LIN {X 0,Y 410.552,Z 311.53,A -85,B 0,C 180,E1 -10538.615,E2 -10538.615} C_VEL
LIN {X 0,Y 410.987,Z 304.76,A -85,B 0,C 180,E1 -10540.095,E2 -10540.095} C_VEL
LIN {X 0,Y 411.569,Z 296.376,A -85,B 0,C 180,E1 -10541.575,E2 -10541.575} C_VEL
LIN {X 0,Y 412.223,Z 287.792,A -85,B 0,C 180,E1 -10542.805,E2 -10542.805} C_VEL
LIN {X 0,Y 412.957,Z 277.054,A -85,B 0,C 180,E1 -10544.052,E2 -10544.052} C_VEL
LIN {X 0,Y 413.773,Z 265.358,A -85,B 0,C 180,E1 -10545.138,E2 -10545.138} C_VEL
LIN {X 0,Y 414.618,Z 253.491,A -85,B 0,C 180,E1 -10545.988,E2 -10545.988} C_VEL
LIN {X 0,Y 414.756,Z 247.262,A -85,B 0,C 180,E1 -10546.361,E2 -10546.361} C_VEL
LIN {X 0,Y 412.907,Z 233.741,A -85,B 0,C 180,E1 -10547.084,E2 -10547.084} C_VEL
LIN {X 0,Y 410.788,Z 220.639,A -85,B 0,C 180,E1 -10547.587,E2 -10547.587} C_VEL
LIN {X 0,Y 410.692,Z 219.451,A -85,B 0,C 180,E1 -10547.631,E2 -10547.631} C_VEL
LIN {X 0,Y 411.028,Z 212.027,A -85,B 0,C 180,E1 -10550.519,E2 -10550.519} C_VEL
LIN {X 0,Y 411.452,Z 202.789,A -85,B 0,C 180,E1 -10554.202,E2 -10554.202} C_VEL
LIN {X 0,Y 411.95,Z 194.811,A -85,B 0,C 180,E1 -10557.484,E2 -10557.484} C_VEL
LIN {X 0,Y 412.504,Z 187.23,A -85,B 0,C 180,E1 -10560.739,E2 -10560.739} C_VEL
LIN {X 0,Y 413.051,Z 181.102,A -85,B 0,C 180,E1 -10563.516,E2 -10563.516} C_VEL
LIN {X 0,Y 413.532,Z 176.073,A -85,B 0,C 180,E1 -10565.897,E2 -10565.897} C_VEL
LIN {X 0,Y 413.222,Z 172.446,A -85,B 0,C 180,E1 -10567.755,E2 -10567.755} C_VEL
LIN {X 0,Y 412.08,Z 166.019,A -85,B 0,C 180,E1 -10571.373,E2 -10571.373} C_VEL
LIN {X 0,Y 411.188,Z 161.268,A -85,B 0,C 180,E1 -10574.489,E2 -10574.489} C_VEL
LIN {X 0,Y 411.182,Z 161.271,A -85,B 0,C 180,E1 -10578.195,E2 -10578.195} C_VEL
LIN {X 0,Y 411.226,Z 161.264,A -85,B 0,C 180,E1 -10580.776,E2 -10580.776} C_VEL
LIN {X 0,Y 411.202,Z 161.267,A -85,B 0,C 180,E1 -10584.471,E2 -10584.471} C_VEL
LIN {X 0,Y 411.211,Z 161.265,A -85,B 0,C 180,E1 -10586.873,E2 -10586.873} C_VEL
LIN {X 0,Y 411.237,Z 161.261,A -85,B 0,C 180,E1 -10590.644,E2 -10590.644} C_VEL
LIN {X 0,Y 411.243,Z 161.26,A -85,B 0,C 180,E1 -10593.619,E2 -10593.619} C_VEL
LIN {X 0,Y 411.208,Z 161.264,A -85,B 0,C 180,E1 -10596.852,E2 -10596.852} C_VEL
LIN {X 0,Y 411.219,Z 161.262,A -85,B 0,C 180,E1 -10600.05,E2 -10600.05} C_VEL
LIN {X 0,Y 411.267,Z 161.257,A -85,B 0,C 180,E1 -10603.131,E2 -10603.131} C_VEL
LIN {X 0,Y 411.31,Z 161.252,A -85,B 0,C 180,E1 -10606.895,E2 -10606.895} C_VEL
LIN {X 0,Y 411.298,Z 161.254,A -85,B 0,C 180,E1 -10610.161,E2 -10610.161} C_VEL
LIN {X 0,Y 411.465,Z 161.233,A -85,B 0,C 180,E1 -10613.133,E2 -10613.133} C_VEL
LIN {X 0,Y 411.315,Z 161.251,A -85,B 0,C 180,E1 -10615.099,E2 -10615.099} C_VEL
LIN {X 0,Y 411.519,Z 161.226,A -85,B 0,C 180,E1 -10618.042,E2 -10618.042} C_VEL
LIN {X 0,Y 411.647,Z 161.211,A -85,B 0,C 180,E1 -10619.999,E2 -10619.999} C_VEL
LIN {X 0,Y 411.469,Z 161.234,A -85,B 0,C 180,E1 -10622.937,E2 -10622.937} C_VEL
LIN {X 0,Y 411.45,Z 161.237,A -85,B 0,C 180,E1 -10626.62,E2 -10626.62} C_VEL
LIN {X 0,Y 411.299,Z 161.255,A -85,B 0,C 180,E1 -10628.846,E2 -10628.846} C_VEL
LIN {X 0,Y 411.065,Z 161.351,A -85,B 0,C 180,E1 -10630.84,E2 -10630.84} C_VEL
LIN {X 0,Y 411.063,Z 163.277,A -85,B 0,C 180,E1 -10632.956,E2 -10632.956} C_VEL
LIN {X 0,Y 410.89,Z 166.763,A -85,B 0,C 180,E1 -10636.695,E2 -10636.695} C_VEL
LIN {X 0,Y 410.695,Z 169.909,A -85,B 0,C 180,E1 -10640.013,E2 -10640.013} C_VEL
LIN {X 0,Y 410.604,Z 172.966,A -85,B 0,C 180,E1 -10643.183,E2 -10643.183} C_VEL
LIN {X 0,Y 410.501,Z 176.153,A -85,B 0,C 180,E1 -10646.431,E2 -10646.431} C_VEL
LIN {X 0,Y 410.553,Z 177.376,A -85,B 0,C 180,E1 -10647.491,E2 -10647.491} C_VEL
LIN {X 0,Y 414.209,Z 190.782,A -85,B 0,C 180,E1 -10648.157,E2 -10648.157} C_VEL
LIN {X 0,Y 415.754,Z 198.207,A -85,B 0,C 180,E1 -10648.593,E2 -10648.593} C_VEL
LIN {X 0,Y 415.142,Z 210.294,A -85,B 0,C 180,E1 -10649.333,E2 -10649.333} C_VEL
LIN {X 0,Y 414.416,Z 221.682,A -85,B 0,C 180,E1 -10650.233,E2 -10650.233} C_VEL
LIN {X 0,Y 413.716,Z 232.745,A -85,B 0,C 180,E1 -10651.345,E2 -10651.345} C_VEL
LIN {X 0,Y 412.965,Z 242.44,A -85,B 0,C 180,E1 -10652.561,E2 -10652.561} C_VEL
LIN {X 0,Y 412.328,Z 250.391,A -85,B 0,C 180,E1 -10653.778,E2 -10653.778} C_VEL
LIN {X 0,Y 411.629,Z 257.985,A -85,B 0,C 180,E1 -10655.195,E2 -10655.195} C_VEL
LIN {X 0,Y 411.155,Z 264.595,A -85,B 0,C 180,E1 -10656.745,E2 -10656.745} C_VEL
LIN {X 0,Y 410.782,Z 269.178,A -85,B 0,C 180,E1 -10658.093,E2 -10658.093} C_VEL
LIN {X 0,Y 410.457,Z 273.169,A -85,B 0,C 180,E1 -10659.6,E2 -10659.6} C_VEL
LIN {X 0,Y 410.255,Z 276.038,A -85,B 0,C 180,E1 -10661.083,E2 -10661.083} C_VEL
LIN {X 0,Y 410.05,Z 277.889,A -85,B 0,C 180,E1 -10662.524,E2 -10662.524} C_VEL
LIN {X 0,Y 409.999,Z 278.849,A -85,B 0,C 180,E1 -10663.95,E2 -10663.95} C_VEL
LIN {X 0,Y 409.939,Z 278.987,A -85,B 0,C 180,E1 -10665.339,E2 -10665.339} C_VEL
LIN {X 0,Y 409.979,Z 278.355,A -85,B 0,C 180,E1 -10666.709,E2 -10666.709} C_VEL
LIN {X 0,Y 410.11,Z 276.96,A -85,B 0,C 180,E1 -10668.061,E2 -10668.061} C_VEL
LIN {X 0,Y 410.276,Z 274.799,A -85,B 0,C 180,E1 -10669.387,E2 -10669.387} C_VEL
LIN {X 0,Y 410.447,Z 271.931,A -85,B 0,C 180,E1 -10670.688,E2 -10670.688} C_VEL
LIN {X 0,Y 410.795,Z 267.236,A -85,B 0,C 180,E1 -10672.293,E2 -10672.293} C_VEL
LIN {X 0,Y 411.226,Z 260.795,A -85,B 0,C 180,E1 -10673.981,E2 -10673.981} C_VEL
LIN {X 0,Y 411.688,Z 253.986,A -85,B 0,C 180,E1 -10675.387,E2 -10675.387} C_VEL
LIN {X 0,Y 412.342,Z 246.022,A -85,B 0,C 180,E1 -10676.723,E2 -10676.723} C_VEL
LIN {X 0,Y 413.027,Z 236.553,A -85,B 0,C 180,E1 -10678.02,E2 -10678.02} C_VEL
LIN {X 0,Y 413.582,Z 227.231,A -85,B 0,C 180,E1 -10679.067,E2 -10679.067} C_VEL
LIN {X 0,Y 414.269,Z 215.745,A -85,B 0,C 180,E1 -10680.102,E2 -10680.102} C_VEL
LIN {X 0,Y 414.955,Z 203.945,A -85,B 0,C 180,E1 -10680.93,E2 -10680.93} C_VEL
LIN {X 0,Y 415.343,Z 197.322,A -85,B 0,C 180,E1 -10681.306,E2 -10681.306} C_VEL
LIN {X 0,Y 412.71,Z 185.249,A -85,B 0,C 180,E1 -10681.972,E2 -10681.972} C_VEL
LIN {X 0,Y 410.376,Z 175.545,A -85,B 0,C 180,E1 -10682.389,E2 -10682.389} C_VEL
LIN {X 0,Y 410.392,Z 171.916,A -85,B 0,C 180,E1 -10685.732,E2 -10685.732} C_VEL
LIN {X 0,Y 410.404,Z 168.584,A -85,B 0,C 180,E1 -10688.923,E2 -10688.923} C_VEL
LIN {X 0,Y 410.492,Z 165.336,A -85,B 0,C 180,E1 -10692.05,E2 -10692.05} C_VEL
LIN {X 0,Y 410.643,Z 162.203,A -85,B 0,C 180,E1 -10695.124,E2 -10695.124} C_VEL
LIN {X 0,Y 410.668,Z 161.335,A -85,B 0,C 180,E1 -10696.137,E2 -10696.137} C_VEL
LIN {X 0,Y 411.106,Z 161.275,A -85,B 0,C 180,E1 -10699.161,E2 -10699.161} C_VEL
LIN {X 0,Y 411.434,Z 161.237,A -85,B 0,C 180,E1 -10702.191,E2 -10702.191} C_VEL
LIN {X 0,Y 411.461,Z 161.234,A -85,B 0,C 180,E1 -10704.118,E2 -10704.118} C_VEL
LIN {X 0,Y 411.511,Z 161.228,A -85,B 0,C 180,E1 -10708.042,E2 -10708.042} C_VEL
LIN {X 0,Y 411.639,Z 161.213,A -85,B 0,C 180,E1 -10710,E2 -10710} C_VEL
LIN {X 0,Y 411.463,Z 161.229,A -85,B 0,C 180,E1 -10712.937,E2 -10712.937} C_VEL
LIN {X 0,Y 411.325,Z 161.247,A -85,B 0,C 180,E1 -10713.48,E2 -10713.48} C_VEL
LIN {X 0,Y 410.551,Z 161.347,A -85,B 0,C 180,E1 -10714.298,E2 -10714.298} C_VEL
LIN {X 0,Y 407.721,Z 161.699,A -85,B 0,C 180,E1 -10715.629,E2 -10715.629} C_VEL
LIN {X 0,Y 405.424,Z 161.983,A -85,B 0,C 180,E1 -10716.704,E2 -10716.704} C_VEL
LIN {X 0,Y 404.482,Z 162.103,A -85,B 0,C 180,E1 -10717.533,E2 -10717.533} C_VEL
LIN {X 0,Y 404.423,Z 162.11,A -85,B 0,C 180,E1 -10717.813,E2 -10717.813} C_VEL
LIN {X 0,Y 404.253,Z 162.131,A -85,B 0,C 180,E1 -10722.041,E2 -10722.041} C_VEL
LIN {X 0,Y 404.203,Z 162.136,A -85,B 0,C 180,E1 -10725.118,E2 -10725.118} C_VEL
LIN {X 0,Y 404.207,Z 162.134,A -85,B 0,C 180,E1 -10728.238,E2 -10728.238} C_VEL
LIN {X 0,Y 404.136,Z 162.146,A -85,B 0,C 180,E1 -10731.419,E2 -10731.419} C_VEL
LIN {X 0,Y 404.174,Z 162.138,A -85,B 0,C 180,E1 -10734.666,E2 -10734.666} C_VEL
LIN {X 0,Y 404.192,Z 162.136,A -85,B 0,C 180,E1 -10738,E2 -10738} C_VEL
LIN {X 0,Y 404.136,Z 162.146,A -85,B 0,C 180,E1 -10741.558,E2 -10741.558} C_VEL
LIN {X 0,Y 404.181,Z 162.14,A -85,B 0,C 180,E1 -10745.016,E2 -10745.016} C_VEL
LIN {X 0,Y 404.153,Z 162.143,A -85,B 0,C 180,E1 -10748.757,E2 -10748.757} C_VEL
LIN {X 0,Y 404.121,Z 162.147,A -85,B 0,C 180,E1 -10751.6,E2 -10751.6} C_VEL
LIN {X 0,Y 404.146,Z 162.142,A -85,B 0,C 180,E1 -10754.523,E2 -10754.523} C_VEL
LIN {X 0,Y 404.134,Z 162.146,A -85,B 0,C 180,E1 -10757.296,E2 -10757.296} C_VEL
LIN {X 0,Y 404.166,Z 162.139,A -85,B 0,C 180,E1 -10759.956,E2 -10759.956} C_VEL
LIN {X 0,Y 404.138,Z 162.145,A -85,B 0,C 180,E1 -10763.125,E2 -10763.125} C_VEL
LIN {X 0,Y 404.143,Z 162.143,A -85,B 0,C 180,E1 -10766.188,E2 -10766.188} C_VEL
LIN {X 0,Y 404.144,Z 162.141,A -85,B 0,C 180,E1 -10769.715,E2 -10769.715} C_VEL
LIN {X 0,Y 404.194,Z 162.137,A -85,B 0,C 180,E1 -10773.123,E2 -10773.123} C_VEL
LIN {X 0,Y 404.176,Z 162.138,A -85,B 0,C 180,E1 -10775.335,E2 -10775.335} C_VEL
LIN {X 0,Y 404.159,Z 162.144,A -85,B 0,C 180,E1 -10778.582,E2 -10778.582} C_VEL
LIN {X 0,Y 404.208,Z 162.135,A -85,B 0,C 180,E1 -10781.762,E2 -10781.762} C_VEL
LIN {X 0,Y 404.206,Z 162.135,A -85,B 0,C 180,E1 -10784.883,E2 -10784.883} C_VEL
LIN {X 0,Y 404.257,Z 162.13,A -85,B 0,C 180,E1 -10787.959,E2 -10787.959} C_VEL
LIN {X 0,Y 404.404,Z 162.114,A -85,B 0,C 180,E1 -10792.131,E2 -10792.131} C_VEL
LIN {X 0,Y 404.419,Z 162.111,A -85,B 0,C 180,E1 -10794.016,E2 -10794.016} C_VEL
LIN {X 0,Y 404.484,Z 162.103,A -85,B 0,C 180,E1 -10798.009,E2 -10798.009} C_VEL
LIN {X 0,Y 404.611,Z 162.087,A -85,B 0,C 180,E1 -10800.001,E2 -10800.001} C_VEL
LIN {X 0,Y 404.417,Z 162.108,A -85,B 0,C 180,E1 -10802.989,E2 -10802.989} C_VEL
LIN {X 0,Y 404.371,Z 162.113,A -85,B 0,C 180,E1 -10806.988,E2 -10806.988} C_VEL
LIN {X 0,Y 404.259,Z 162.131,A -85,B 0,C 180,E1 -10810.012,E2 -10810.012} C_VEL
LIN {X 0,Y 404.268,Z 162.128,A -85,B 0,C 180,E1 -10813.212,E2 -10813.212} C_VEL
LIN {X 0,Y 404.218,Z 162.133,A -85,B 0,C 180,E1 -10817.007,E2 -10817.007} C_VEL
LIN {X 0,Y 404.166,Z 162.139,A -85,B 0,C 180,E1 -10820.352,E2 -10820.352} C_VEL
LIN {X 0,Y 404.172,Z 162.142,A -85,B 0,C 180,E1 -10823.575,E2 -10823.575} C_VEL
LIN {X 0,Y 404.186,Z 162.139,A -85,B 0,C 180,E1 -10825.767,E2 -10825.767} C_VEL
LIN {X 0,Y 404.197,Z 162.137,A -85,B 0,C 180,E1 -10828,E2 -10828} C_VEL
LIN {X 0,Y 404.141,Z 162.146,A -85,B 0,C 180,E1 -10831.558,E2 -10831.558} C_VEL
LIN {X 0,Y 404.186,Z 162.14,A -85,B 0,C 180,E1 -10835.017,E2 -10835.017} C_VEL
LIN {X 0,Y 404.155,Z 162.142,A -85,B 0,C 180,E1 -10838.757,E2 -10838.757} C_VEL
LIN {X 0,Y 404.125,Z 162.146,A -85,B 0,C 180,E1 -10841.6,E2 -10841.6} C_VEL
LIN {X 0,Y 404.148,Z 162.138,A -85,B 0,C 180,E1 -10844.522,E2 -10844.522} C_VEL
LIN {X 0,Y 404.174,Z 162.299,A -85,B 0,C 180,E1 -10846.103,E2 -10846.103} C_VEL
LIN {X 0,Y 405.082,Z 167.107,A -85,B 0,C 180,E1 -10848.755,E2 -10848.755} C_VEL
LIN {X 0,Y 406.218,Z 173.548,A -85,B 0,C 180,E1 -10852.108,E2 -10852.108} C_VEL
LIN {X 0,Y 406.527,Z 177.404,A -85,B 0,C 180,E1 -10854,E2 -10854} C_VEL
LIN {X 0,Y 406.009,Z 183.846,A -85,B 0,C 180,E1 -10856.957,E2 -10856.957} C_VEL
LIN {X 0,Y 405.458,Z 190.289,A -85,B 0,C 180,E1 -10859.823,E2 -10859.823} C_VEL
LIN {X 0,Y 404.993,Z 196.978,A -85,B 0,C 180,E1 -10862.704,E2 -10862.704} C_VEL
LIN {X 0,Y 404.383,Z 205.889,A -85,B 0,C 180,E1 -10866.439,E2 -10866.439} C_VEL
LIN {X 0,Y 403.91,Z 214.589,A -85,B 0,C 180,E1 -10869.985,E2 -10869.985} C_VEL
LIN {X 0,Y 403.652,Z 219.873,A -85,B 0,C 180,E1 -10872.097,E2 -10872.097} C_VEL
LIN {X 0,Y 405.923,Z 233.642,A -85,B 0,C 180,E1 -10872.623,E2 -10872.623} C_VEL
LIN {X 0,Y 407.729,Z 246.619,A -85,B 0,C 180,E1 -10873.319,E2 -10873.319} C_VEL
LIN {X 0,Y 407.879,Z 251.732,A -85,B 0,C 180,E1 -10873.631,E2 -10873.631} C_VEL
LIN {X 0,Y 407.03,Z 263.745,A -85,B 0,C 180,E1 -10874.477,E2 -10874.477} C_VEL
LIN {X 0,Y 406.19,Z 275.278,A -85,B 0,C 180,E1 -10875.522,E2 -10875.522} C_VEL
LIN {X 0,Y 405.413,Z 285.747,A -85,B 0,C 180,E1 -10876.721,E2 -10876.721} C_VEL
LIN {X 0,Y 404.71,Z 294.651,A -85,B 0,C 180,E1 -10877.972,E2 -10877.972} C_VEL
LIN {X 0,Y 404.038,Z 303.354,A -85,B 0,C 180,E1 -10879.476,E2 -10879.476} C_VEL
LIN {X 0,Y 403.575,Z 310.309,A -85,B 0,C 180,E1 -10880.983,E2 -10880.983} C_VEL
LIN {X 0,Y 403.204,Z 315.883,A -85,B 0,C 180,E1 -10882.488,E2 -10882.488} C_VEL
LIN {X 0,Y 403.016,Z 320.261,A -85,B 0,C 180,E1 -10883.994,E2 -10883.994} C_VEL
LIN {X 0,Y 403.002,Z 322.579,A -85,B 0,C 180,E1 -10884.998,E2 -10884.998} C_VEL
LIN {X 0,Y 402.876,Z 324.452,A -85,B 0,C 180,E1 -10885.999,E2 -10885.999} C_VEL
LIN {X 0,Y 402.895,Z 325.862,A -85,B 0,C 180,E1 -10887,E2 -10887} C_VEL
LIN {X 0,Y 402.92,Z 326.863,A -85,B 0,C 180,E1 -10888.001,E2 -10888.001} C_VEL
LIN {X 0,Y 402.879,Z 327.673,A -85,B 0,C 180,E1 -10890,E2 -10890} C_VEL
LIN {X 0,Y 402.875,Z 327.442,A -85,B 0,C 180,E1 -10891,E2 -10891} C_VEL
LIN {X 0,Y 402.922,Z 326.814,A -85,B 0,C 180,E1 -10891.999,E2 -10891.999} C_VEL
LIN {X 0,Y 402.909,Z 325.788,A -85,B 0,C 180,E1 -10893,E2 -10893} C_VEL
LIN {X 0,Y 402.878,Z 324.353,A -85,B 0,C 180,E1 -10894.001,E2 -10894.001} C_VEL
LIN {X 0,Y 403.007,Z 321.356,A -85,B 0,C 180,E1 -10895.504,E2 -10895.504} C_VEL
LIN {X 0,Y 403.118,Z 317.303,A -85,B 0,C 180,E1 -10897.01,E2 -10897.01} C_VEL
LIN {X 0,Y 403.518,Z 311.093,A -85,B 0,C 180,E1 -10898.766,E2 -10898.766} C_VEL
LIN {X 0,Y 403.962,Z 304.323,A -85,B 0,C 180,E1 -10900.272,E2 -10900.272} C_VEL
LIN {X 0,Y 404.576,Z 295.944,A -85,B 0,C 180,E1 -10901.778,E2 -10901.778} C_VEL
LIN {X 0,Y 405.244,Z 287.368,A -85,B 0,C 180,E1 -10903.03,E2 -10903.03} C_VEL
LIN {X 0,Y 405.982,Z 277.521,A -85,B 0,C 180,E1 -10904.204,E2 -10904.204} C_VEL
LIN {X 0,Y 406.781,Z 266.392,A -85,B 0,C 180,E1 -10905.277,E2 -10905.277} C_VEL
LIN {X 0,Y 407.649,Z 255.13,A -85,B 0,C 180,E1 -10906.134,E2 -10906.134} C_VEL
LIN {X 0,Y 407.91,Z 248.55,A -85,B 0,C 180,E1 -10906.55,E2 -10906.55} C_VEL
LIN {X 0,Y 406.128,Z 235.006,A -85,B 0,C 180,E1 -10907.314,E2 -10907.314} C_VEL
LIN {X 0,Y 404.092,Z 222.004,A -85,B 0,C 180,E1 -10907.858,E2 -10907.858} C_VEL
LIN {X 0,Y 403.633,Z 218.99,A -85,B 0,C 180,E1 -10907.97,E2 -10907.97} C_VEL
LIN {X 0,Y 403.958,Z 211.643,A -85,B 0,C 180,E1 -10910.895,E2 -10910.895} C_VEL
LIN {X 0,Y 404.447,Z 202.456,A -85,B 0,C 180,E1 -10914.648,E2 -10914.648} C_VEL
LIN {X 0,Y 404.985,Z 194.699,A -85,B 0,C 180,E1 -10917.941,E2 -10917.941} C_VEL
LIN {X 0,Y 405.601,Z 187.044,A -85,B 0,C 180,E1 -10921.321,E2 -10921.321} C_VEL
LIN {X 0,Y 406.306,Z 179.599,A -85,B 0,C 180,E1 -10924.807,E2 -10924.807} C_VEL
LIN {X 0,Y 406.507,Z 175.952,A -85,B 0,C 180,E1 -10926.617,E2 -10926.617} C_VEL
LIN {X 0,Y 405.925,Z 171.895,A -85,B 0,C 180,E1 -10928.82,E2 -10928.82} C_VEL
LIN {X 0,Y 405.039,Z 166.908,A -85,B 0,C 180,E1 -10931.745,E2 -10931.745} C_VEL
LIN {X 0,Y 404.129,Z 162.148,A -85,B 0,C 180,E1 -10934.912,E2 -10934.912} C_VEL
LIN {X 0,Y 404.141,Z 162.149,A -85,B 0,C 180,E1 -10937.296,E2 -10937.296} C_VEL
LIN {X 0,Y 404.173,Z 162.145,A -85,B 0,C 180,E1 -10939.955,E2 -10939.955} C_VEL
LIN {X 0,Y 404.141,Z 162.147,A -85,B 0,C 180,E1 -10943.125,E2 -10943.125} C_VEL
LIN {X 0,Y 404.149,Z 162.144,A -85,B 0,C 180,E1 -10946.188,E2 -10946.188} C_VEL
LIN {X 0,Y 404.15,Z 162.144,A -85,B 0,C 180,E1 -10949.715,E2 -10949.715} C_VEL
LIN {X 0,Y 404.2,Z 162.136,A -85,B 0,C 180,E1 -10953.123,E2 -10953.123} C_VEL
LIN {X 0,Y 404.182,Z 162.138,A -85,B 0,C 180,E1 -10955.334,E2 -10955.334} C_VEL
LIN {X 0,Y 404.143,Z 162.146,A -85,B 0,C 180,E1 -10958.58,E2 -10958.58} C_VEL
LIN {X 0,Y 404.209,Z 162.133,A -85,B 0,C 180,E1 -10961.761,E2 -10961.761} C_VEL
LIN {X 0,Y 404.211,Z 162.136,A -85,B 0,C 180,E1 -10964.882,E2 -10964.882} C_VEL
LIN {X 0,Y 404.261,Z 162.13,A -85,B 0,C 180,E1 -10967.958,E2 -10967.958} C_VEL
LIN {X 0,Y 404.438,Z 162.108,A -85,B 0,C 180,E1 -10972.099,E2 -10972.099} C_VEL
LIN {X 0,Y 404.428,Z 162.109,A -85,B 0,C 180,E1 -10974.015,E2 -10974.015} C_VEL
LIN {X 0,Y 404.487,Z 162.102,A -85,B 0,C 180,E1 -10978.008,E2 -10978.008} C_VEL
LIN {X 0,Y 404.616,Z 162.087,A -85,B 0,C 180,E1 -10979.999,E2 -10979.999} C_VEL
LIN {X 0,Y 404.426,Z 162.111,A -85,B 0,C 180,E1 -10982.988,E2 -10982.988} C_VEL
LIN {X 0,Y 404.395,Z 162.115,A -85,B 0,C 180,E1 -10986.619,E2 -10986.619} C_VEL
LIN {X 0,Y 404.239,Z 162.134,A -85,B 0,C 180,E1 -10989.002,E2 -10989.002} C_VEL
LIN {X 0,Y 404.05,Z 162.548,A -85,B 0,C 180,E1 -10991.03,E2 -10991.03} C_VEL
LIN {X 0,Y 403.942,Z 165.314,A -85,B 0,C 180,E1 -10994.097,E2 -10994.097} C_VEL
LIN {X 0,Y 403.8,Z 168.179,A -85,B 0,C 180,E1 -10997.21,E2 -10997.21} C_VEL
LIN {X 0,Y 403.637,Z 171.148,A -85,B 0,C 180,E1 -11000.379,E2 -11000.379} C_VEL
LIN {X 0,Y 403.533,Z 174.235,A -85,B 0,C 180,E1 -11003.613,E2 -11003.613} C_VEL
LIN {X 0,Y 403.457,Z 177.672,A -85,B 0,C 180,E1 -11007.138,E2 -11007.138} C_VEL
LIN {X 0,Y 407.287,Z 191.331,A -85,B 0,C 180,E1 -11007.845,E2 -11007.845} C_VEL
LIN {X 0,Y 408.819,Z 198.299,A -85,B 0,C 180,E1 -11008.268,E2 -11008.268} C_VEL
LIN {X 0,Y 408.404,Z 210.267,A -85,B 0,C 180,E1 -11009.016,E2 -11009.016} C_VEL
LIN {X 0,Y 407.575,Z 222.551,A -85,B 0,C 180,E1 -11010.003,E2 -11010.003} C_VEL
LIN {X 0,Y 406.873,Z 233.199,A -85,B 0,C 180,E1 -11011.097,E2 -11011.097} C_VEL
LIN {X 0,Y 406.159,Z 241.938,A -85,B 0,C 180,E1 -11012.197,E2 -11012.197} C_VEL
LIN {X 0,Y 405.346,Z 251.431,A -85,B 0,C 180,E1 -11013.67,E2 -11013.67} C_VEL
LIN {X 0,Y 404.561,Z 259.614,A -85,B 0,C 180,E1 -11015.265,E2 -11015.265} C_VEL
LIN {X 0,Y 404.076,Z 266.026,A -85,B 0,C 180,E1 -11016.863,E2 -11016.863} C_VEL
LIN {X 0,Y 403.659,Z 270.92,A -85,B 0,C 180,E1 -11018.419,E2 -11018.419} C_VEL
LIN {X 0,Y 403.308,Z 274.978,A -85,B 0,C 180,E1 -11020.147,E2 -11020.147} C_VEL
LIN {X 0,Y 403.125,Z 277.173,A -85,B 0,C 180,E1 -11021.489,E2 -11021.489} C_VEL
LIN {X 0,Y 402.937,Z 278.69,A -85,B 0,C 180,E1 -11022.898,E2 -11022.898} C_VEL
LIN {X 0,Y 402.879,Z 279.416,A -85,B 0,C 180,E1 -11024.338,E2 -11024.338} C_VEL
LIN {X 0,Y 402.864,Z 279.33,A -85,B 0,C 180,E1 -11025.749,E2 -11025.749} C_VEL
LIN {X 0,Y 402.937,Z 278.433,A -85,B 0,C 180,E1 -11027.138,E2 -11027.138} C_VEL
LIN {X 0,Y 403.094,Z 276.709,A -85,B 0,C 180,E1 -11028.564,E2 -11028.564} C_VEL
LIN {X 0,Y 403.296,Z 273.981,A -85,B 0,C 180,E1 -11030.063,E2 -11030.063} C_VEL
LIN {X 0,Y 403.55,Z 270.13,A -85,B 0,C 180,E1 -11031.599,E2 -11031.599} C_VEL
LIN {X 0,Y 403.924,Z 264.993,A -85,B 0,C 180,E1 -11033.164,E2 -11033.164} C_VEL
LIN {X 0,Y 404.415,Z 258.326,A -85,B 0,C 180,E1 -11034.762,E2 -11034.762} C_VEL
LIN {X 0,Y 405.074,Z 249.676,A -85,B 0,C 180,E1 -11036.386,E2 -11036.386} C_VEL
LIN {X 0,Y 405.865,Z 240.146,A -85,B 0,C 180,E1 -11037.816,E2 -11037.816} C_VEL
LIN {X 0,Y 406.542,Z 230.234,A -85,B 0,C 180,E1 -11039.011,E2 -11039.011} C_VEL
LIN {X 0,Y 407.239,Z 218.894,A -85,B 0,C 180,E1 -11040.111,E2 -11040.111} C_VEL
LIN {X 0,Y 408,Z 206.876,A -85,B 0,C 180,E1 -11041.022,E2 -11041.022} C_VEL
LIN {X 0,Y 408.289,Z 197.054,A -85,B 0,C 180,E1 -11041.612,E2 -11041.612} C_VEL
LIN {X 0,Y 405.302,Z 183.991,A -85,B 0,C 180,E1 -11042.329,E2 -11042.329} C_VEL
LIN {X 0,Y 403.301,Z 175.836,A -85,B 0,C 180,E1 -11042.713,E2 -11042.713} C_VEL
LIN {X 0,Y 403.374,Z 173.101,A -85,B 0,C 180,E1 -11045.282,E2 -11045.282} C_VEL
LIN {X 0,Y 403.32,Z 169.729,A -85,B 0,C 180,E1 -11048.535,E2 -11048.535} C_VEL
LIN {X 0,Y 403.441,Z 166.434,A -85,B 0,C 180,E1 -11051.726,E2 -11051.726} C_VEL
LIN {X 0,Y 403.567,Z 163.266,A -85,B 0,C 180,E1 -11054.857,E2 -11054.857} C_VEL
LIN {X 0,Y 403.584,Z 162.249,A -85,B 0,C 180,E1 -11055.889,E2 -11055.889} C_VEL
LIN {X 0,Y 404.027,Z 162.157,A -85,B 0,C 180,E1 -11058.969,E2 -11058.969} C_VEL
LIN {X 0,Y 404.374,Z 162.117,A -85,B 0,C 180,E1 -11062.157,E2 -11062.157} C_VEL
LIN {X 0,Y 404.408,Z 162.113,A -85,B 0,C 180,E1 -11064.015,E2 -11064.015} C_VEL
LIN {X 0,Y 404.48,Z 162.104,A -85,B 0,C 180,E1 -11068.008,E2 -11068.008} C_VEL
LIN {X 0,Y 404.608,Z 162.089,A -85,B 0,C 180,E1 -11070,E2 -11070} C_VEL
LIN {X 0,Y 404.42,Z 162.107,A -85,B 0,C 180,E1 -11072.988,E2 -11072.988} C_VEL
LIN {X 0,Y 404.406,Z 162.109,A -85,B 0,C 180,E1 -11076.987,E2 -11076.987} C_VEL
LIN {X 0,Y 404.423,Z 162.11,A -85,B 0,C 180,E1 -11077.813,E2 -11077.813} C_VEL
LIN {X 0,Y 403.774,Z 162.195,A -85,B 0,C 180,E1 -11078.644,E2 -11078.644} C_VEL
LIN {X 0,Y 400.822,Z 162.56,A -85,B 0,C 180,E1 -11079.99,E2 -11079.99} C_VEL
LIN {X 0,Y 398.32,Z 162.868,A -85,B 0,C 180,E1 -11081.078,E2 -11081.078} C_VEL
LIN {X 0,Y 397.278,Z 163.001,A -85,B 0,C 180,E1 -11081.921,E2 -11081.921} C_VEL
LIN {X 0,Y 397.212,Z 163.006,A -85,B 0,C 180,E1 -11082.207,E2 -11082.207} C_VEL
LIN {X 0,Y 397.176,Z 163.012,A -85,B 0,C 180,E1 -11085.392,E2 -11085.392} C_VEL
LIN {X 0,Y 397.159,Z 163.011,A -85,B 0,C 180,E1 -11088.573,E2 -11088.573} C_VEL
LIN {X 0,Y 397.094,Z 163.023,A -85,B 0,C 180,E1 -11091.819,E2 -11091.819} C_VEL
LIN {X 0,Y 397.153,Z 163.015,A -85,B 0,C 180,E1 -11095.132,E2 -11095.132} C_VEL
LIN {X 0,Y 397.158,Z 163.014,A -85,B 0,C 180,E1 -11097.776,E2 -11097.776} C_VEL
LIN {X 0,Y 397.075,Z 163.024,A -85,B 0,C 180,E1 -11100.883,E2 -11100.883} C_VEL
LIN {X 0,Y 397.122,Z 163.016,A -85,B 0,C 180,E1 -11104.494,E2 -11104.494} C_VEL
LIN {X 0,Y 397.1,Z 163.019,A -85,B 0,C 180,E1 -11108.275,E2 -11108.275} C_VEL
LIN {X 0,Y 397.086,Z 163.024,A -85,B 0,C 180,E1 -11110.909,E2 -11110.909} C_VEL
LIN {X 0,Y 397.101,Z 163.02,A -85,B 0,C 180,E1 -11113.648,E2 -11113.648} C_VEL
LIN {X 0,Y 397.1,Z 163.021,A -85,B 0,C 180,E1 -11116.521,E2 -11116.521} C_VEL
LIN {X 0,Y 397.112,Z 163.019,A -85,B 0,C 180,E1 -11120.423,E2 -11120.423} C_VEL
LIN {X 0,Y 397.107,Z 163.019,A -85,B 0,C 180,E1 -11124.266,E2 -11124.266} C_VEL
LIN {X 0,Y 397.113,Z 163.022,A -85,B 0,C 180,E1 -11126.728,E2 -11126.728} C_VEL
LIN {X 0,Y 397.123,Z 163.018,A -85,B 0,C 180,E1 -11130.296,E2 -11130.296} C_VEL
LIN {X 0,Y 397.193,Z 163.012,A -85,B 0,C 180,E1 -11132.61,E2 -11132.61} C_VEL
LIN {X 0,Y 397.132,Z 163.016,A -85,B 0,C 180,E1 -11135.982,E2 -11135.982} C_VEL
LIN {X 0,Y 397.138,Z 163.014,A -85,B 0,C 180,E1 -11139.705,E2 -11139.705} C_VEL
LIN {X 0,Y 397.182,Z 163.011,A -85,B 0,C 180,E1 -11142.845,E2 -11142.845} C_VEL
LIN {X 0,Y 397.229,Z 163.006,A -85,B 0,C 180,E1 -11146.703,E2 -11146.703} C_VEL
LIN {X 0,Y 397.218,Z 163.006,A -85,B 0,C 180,E1 -11149.81,E2 -11149.81} C_VEL
LIN {X 0,Y 397.343,Z 162.99,A -85,B 0,C 180,E1 -11152.888,E2 -11152.888} C_VEL
LIN {X 0,Y 397.255,Z 163,A -85,B 0,C 180,E1 -11154.926,E2 -11154.926} C_VEL
LIN {X 0,Y 397.453,Z 162.979,A -85,B 0,C 180,E1 -11157.974,E2 -11157.974} C_VEL
LIN {X 0,Y 397.58,Z 162.963,A -85,B 0,C 180,E1 -11160.001,E2 -11160.001} C_VEL
LIN {X 0,Y 397.377,Z 162.985,A -85,B 0,C 180,E1 -11163.042,E2 -11163.042} C_VEL
LIN {X 0,Y 397.347,Z 162.992,A -85,B 0,C 180,E1 -11166.092,E2 -11166.092} C_VEL
LIN {X 0,Y 397.237,Z 163.003,A -85,B 0,C 180,E1 -11169.163,E2 -11169.163} C_VEL
LIN {X 0,Y 397.221,Z 163.006,A -85,B 0,C 180,E1 -11172.259,E2 -11172.259} C_VEL
LIN {X 0,Y 397.181,Z 163.012,A -85,B 0,C 180,E1 -11175.392,E2 -11175.392} C_VEL
LIN {X 0,Y 397.164,Z 163.011,A -85,B 0,C 180,E1 -11178.574,E2 -11178.574} C_VEL
LIN {X 0,Y 397.099,Z 163.023,A -85,B 0,C 180,E1 -11181.819,E2 -11181.819} C_VEL
LIN {X 0,Y 397.159,Z 163.015,A -85,B 0,C 180,E1 -11185.132,E2 -11185.132} C_VEL
LIN {X 0,Y 397.164,Z 163.014,A -85,B 0,C 180,E1 -11187.776,E2 -11187.776} C_VEL
LIN {X 0,Y 397.081,Z 163.023,A -85,B 0,C 180,E1 -11190.883,E2 -11190.883} C_VEL
LIN {X 0,Y 397.127,Z 163.016,A -85,B 0,C 180,E1 -11194.494,E2 -11194.494} C_VEL
LIN {X 0,Y 397.103,Z 163.021,A -85,B 0,C 180,E1 -11198.275,E2 -11198.275} C_VEL
LIN {X 0,Y 397.091,Z 163.024,A -85,B 0,C 180,E1 -11200.909,E2 -11200.909} C_VEL
LIN {X 0,Y 397.103,Z 163.017,A -85,B 0,C 180,E1 -11203.649,E2 -11203.649} C_VEL
LIN {X 0,Y 397.136,Z 163.143,A -85,B 0,C 180,E1 -11205.735,E2 -11205.735} C_VEL
LIN {X 0,Y 398.322,Z 169.624,A -85,B 0,C 180,E1 -11209.35,E2 -11209.35} C_VEL
LIN {X 0,Y 399.32,Z 175.375,A -85,B 0,C 180,E1 -11212.373,E2 -11212.373} C_VEL
LIN {X 0,Y 399.471,Z 179.726,A -85,B 0,C 180,E1 -11214.509,E2 -11214.509} C_VEL
LIN {X 0,Y 398.826,Z 187.422,A -85,B 0,C 180,E1 -11218.086,E2 -11218.086} C_VEL
LIN {X 0,Y 398.083,Z 196.18,A -85,B 0,C 180,E1 -11221.974,E2 -11221.974} C_VEL
LIN {X 0,Y 397.458,Z 204.267,A -85,B 0,C 180,E1 -11225.447,E2 -11225.447} C_VEL
LIN {X 0,Y 396.996,Z 212.055,A -85,B 0,C 180,E1 -11228.721,E2 -11228.721} C_VEL
LIN {X 0,Y 396.624,Z 219.652,A -85,B 0,C 180,E1 -11231.785,E2 -11231.785} C_VEL
LIN {X 0,Y 398.928,Z 233.436,A -85,B 0,C 180,E1 -11232.325,E2 -11232.325} C_VEL
LIN {X 0,Y 400.743,Z 246.734,A -85,B 0,C 180,E1 -11233.059,E2 -11233.059} C_VEL
LIN {X 0,Y 401.032,Z 251.525,A -85,B 0,C 180,E1 -11233.365,E2 -11233.365} C_VEL
LIN {X 0,Y 400.161,Z 263.232,A -85,B 0,C 180,E1 -11234.203,E2 -11234.203} C_VEL
LIN {X 0,Y 399.27,Z 274.788,A -85,B 0,C 180,E1 -11235.265,E2 -11235.265} C_VEL
LIN {X 0,Y 398.478,Z 285.337,A -85,B 0,C 180,E1 -11236.494,E2 -11236.494} C_VEL
LIN {X 0,Y 397.747,Z 294.191,A -85,B 0,C 180,E1 -11237.759,E2 -11237.759} C_VEL
LIN {X 0,Y 396.992,Z 302.906,A -85,B 0,C 180,E1 -11239.288,E2 -11239.288} C_VEL
LIN {X 0,Y 396.499,Z 309.87,A -85,B 0,C 180,E1 -11240.821,E2 -11240.821} C_VEL
LIN {X 0,Y 396.139,Z 315.453,A -85,B 0,C 180,E1 -11242.354,E2 -11242.354} C_VEL
LIN {X 0,Y 395.951,Z 319.837,A -85,B 0,C 180,E1 -11243.887,E2 -11243.887} C_VEL
LIN {X 0,Y 395.915,Z 322.156,A -85,B 0,C 180,E1 -11244.908,E2 -11244.908} C_VEL
LIN {X 0,Y 395.801,Z 324.032,A -85,B 0,C 180,E1 -11245.927,E2 -11245.927} C_VEL
LIN {X 0,Y 395.799,Z 325.443,A -85,B 0,C 180,E1 -11246.947,E2 -11246.947} C_VEL
LIN {X 0,Y 395.853,Z 326.445,A -85,B 0,C 180,E1 -11247.965,E2 -11247.965} C_VEL
LIN {X 0,Y 395.805,Z 327.255,A -85,B 0,C 180,E1 -11250,E2 -11250} C_VEL
LIN {X 0,Y 395.804,Z 327.024,A -85,B 0,C 180,E1 -11251.018,E2 -11251.018} C_VEL
LIN {X 0,Y 395.855,Z 326.395,A -85,B 0,C 180,E1 -11252.035,E2 -11252.035} C_VEL
LIN {X 0,Y 395.812,Z 325.366,A -85,B 0,C 180,E1 -11253.054,E2 -11253.054} C_VEL
LIN {X 0,Y 395.803,Z 323.931,A -85,B 0,C 180,E1 -11254.073,E2 -11254.073} C_VEL
LIN {X 0,Y 395.908,Z 320.932,A -85,B 0,C 180,E1 -11255.603,E2 -11255.603} C_VEL
LIN {X 0,Y 396.063,Z 316.881,A -85,B 0,C 180,E1 -11257.135,E2 -11257.135} C_VEL
LIN {X 0,Y 396.459,Z 310.672,A -85,B 0,C 180,E1 -11258.923,E2 -11258.923} C_VEL
LIN {X 0,Y 396.913,Z 303.901,A -85,B 0,C 180,E1 -11260.457,E2 -11260.457} C_VEL
LIN {X 0,Y 397.569,Z 295.523,A -85,B 0,C 180,E1 -11261.988,E2 -11261.988} C_VEL
LIN {X 0,Y 398.29,Z 286.963,A -85,B 0,C 180,E1 -11263.261,E2 -11263.261} C_VEL
LIN {X 0,Y 399.098,Z 276.659,A -85,B 0,C 180,E1 -11264.507,E2 -11264.507} C_VEL
LIN {X 0,Y 399.932,Z 266.039,A -85,B 0,C 180,E1 -11265.545,E2 -11265.545} C_VEL
LIN {X 0,Y 400.816,Z 254.893,A -85,B 0,C 180,E1 -11266.412,E2 -11266.412} C_VEL
LIN {X 0,Y 401.054,Z 249.628,A -85,B 0,C 180,E1 -11266.757,E2 -11266.757} C_VEL
LIN {X 0,Y 399.451,Z 236.896,A -85,B 0,C 180,E1 -11267.522,E2 -11267.522} C_VEL
LIN {X 0,Y 397.384,Z 223.179,A -85,B 0,C 180,E1 -11268.138,E2 -11268.138} C_VEL
LIN {X 0,Y 396.601,Z 218.502,A -85,B 0,C 180,E1 -11268.333,E2 -11268.333} C_VEL
LIN {X 0,Y 396.922,Z 211.273,A -85,B 0,C 180,E1 -11271.283,E2 -11271.283} C_VEL
LIN {X 0,Y 397.377,Z 203.436,A -85,B 0,C 180,E1 -11274.559,E2 -11274.559} C_VEL
LIN {X 0,Y 397.96,Z 195.512,A -85,B 0,C 180,E1 -11277.992,E2 -11277.992} C_VEL
LIN {X 0,Y 398.738,Z 186.834,A -85,B 0,C 180,E1 -11281.923,E2 -11281.923} C_VEL
LIN {X 0,Y 399.457,Z 179.434,A -85,B 0,C 180,E1 -11285.493,E2 -11285.493} C_VEL
LIN {X 0,Y 399.524,Z 177.06,A -85,B 0,C 180,E1 -11286.734,E2 -11286.734} C_VEL
LIN {X 0,Y 398.777,Z 172.339,A -85,B 0,C 180,E1 -11289.38,E2 -11289.38} C_VEL
LIN {X 0,Y 397.995,Z 167.765,A -85,B 0,C 180,E1 -11292.147,E2 -11292.147} C_VEL
LIN {X 0,Y 397.105,Z 163.024,A -85,B 0,C 180,E1 -11295.379,E2 -11295.379} C_VEL
LIN {X 0,Y 397.093,Z 163.027,A -85,B 0,C 180,E1 -11299.091,E2 -11299.091} C_VEL
LIN {X 0,Y 397.108,Z 163.024,A -85,B 0,C 180,E1 -11301.725,E2 -11301.725} C_VEL
LIN {X 0,Y 397.13,Z 163.017,A -85,B 0,C 180,E1 -11305.507,E2 -11305.507} C_VEL
LIN {X 0,Y 397.083,Z 163.023,A -85,B 0,C 180,E1 -11309.117,E2 -11309.117} C_VEL
LIN {X 0,Y 397.199,Z 163.009,A -85,B 0,C 180,E1 -11312.61,E2 -11312.61} C_VEL
LIN {X 0,Y 397.137,Z 163.017,A -85,B 0,C 180,E1 -11315.982,E2 -11315.982} C_VEL
LIN {X 0,Y 397.143,Z 163.014,A -85,B 0,C 180,E1 -11319.704,E2 -11319.704} C_VEL
LIN {X 0,Y 397.186,Z 163.011,A -85,B 0,C 180,E1 -11322.845,E2 -11322.845} C_VEL
LIN {X 0,Y 397.233,Z 163.006,A -85,B 0,C 180,E1 -11326.702,E2 -11326.702} C_VEL
LIN {X 0,Y 397.222,Z 163.008,A -85,B 0,C 180,E1 -11329.809,E2 -11329.809} C_VEL
LIN {X 0,Y 397.369,Z 162.989,A -85,B 0,C 180,E1 -11332.888,E2 -11332.888} C_VEL
LIN {X 0,Y 397.259,Z 163.002,A -85,B 0,C 180,E1 -11334.925,E2 -11334.925} C_VEL
LIN {X 0,Y 397.456,Z 162.978,A -85,B 0,C 180,E1 -11337.973,E2 -11337.973} C_VEL
LIN {X 0,Y 397.585,Z 162.963,A -85,B 0,C 180,E1 -11339.999,E2 -11339.999} C_VEL
LIN {X 0,Y 397.384,Z 162.988,A -85,B 0,C 180,E1 -11343.041,E2 -11343.041} C_VEL
LIN {X 0,Y 397.345,Z 162.993,A -85,B 0,C 180,E1 -11346.615,E2 -11346.615} C_VEL
LIN {X 0,Y 397.173,Z 163.014,A -85,B 0,C 180,E1 -11349.163,E2 -11349.163} C_VEL
LIN {X 0,Y 397.072,Z 163.029,A -85,B 0,C 180,E1 -11350.194,E2 -11350.194} C_VEL
LIN {X 0,Y 396.998,Z 165.589,A -85,B 0,C 180,E1 -11353.305,E2 -11353.305} C_VEL
LIN {X 0,Y 396.787,Z 168.887,A -85,B 0,C 180,E1 -11356.968,E2 -11356.968} C_VEL
LIN {X 0,Y 396.56,Z 172.412,A -85,B 0,C 180,E1 -11360.759,E2 -11360.759} C_VEL
LIN {X 0,Y 396.453,Z 175.535,A -85,B 0,C 180,E1 -11364.061,E2 -11364.061} C_VEL
LIN {X 0,Y 396.417,Z 178.136,A -85,B 0,C 180,E1 -11366.77,E2 -11366.77} C_VEL
LIN {X 0,Y 400.565,Z 192.844,A -85,B 0,C 180,E1 -11367.575,E2 -11367.575} C_VEL
LIN {X 0,Y 402.162,Z 200.663,A -85,B 0,C 180,E1 -11368.075,E2 -11368.075} C_VEL
LIN {X 0,Y 401.555,Z 211.931,A -85,B 0,C 180,E1 -11368.807,E2 -11368.807} C_VEL
LIN {X 0,Y 400.807,Z 222.671,A -85,B 0,C 180,E1 -11369.692,E2 -11369.692} C_VEL
LIN {X 0,Y 400.093,Z 233.095,A -85,B 0,C 180,E1 -11370.77,E2 -11370.77} C_VEL
LIN {X 0,Y 399.205,Z 243.228,A -85,B 0,C 180,E1 -11372.077,E2 -11372.077} C_VEL
LIN {X 0,Y 398.382,Z 252.323,A -85,B 0,C 180,E1 -11373.532,E2 -11373.532} C_VEL
LIN {X 0,Y 397.617,Z 259.675,A -85,B 0,C 180,E1 -11374.988,E2 -11374.988} C_VEL
LIN {X 0,Y 397.074,Z 266.394,A -85,B 0,C 180,E1 -11376.68,E2 -11376.68} C_VEL
LIN {X 0,Y 396.608,Z 271.489,A -85,B 0,C 180,E1 -11378.331,E2 -11378.331} C_VEL
LIN {X 0,Y 396.336,Z 274.656,A -85,B 0,C 180,E1 -11379.669,E2 -11379.669} C_VEL
LIN {X 0,Y 396.12,Z 277.09,A -85,B 0,C 180,E1 -11381.029,E2 -11381.029} C_VEL
LIN {X 0,Y 395.907,Z 278.782,A -85,B 0,C 180,E1 -11382.419,E2 -11382.419} C_VEL
LIN {X 0,Y 395.798,Z 279.699,A -85,B 0,C 180,E1 -11383.828,E2 -11383.828} C_VEL
LIN {X 0,Y 395.76,Z 279.863,A -85,B 0,C 180,E1 -11385.261,E2 -11385.261} C_VEL
LIN {X 0,Y 395.806,Z 279.226,A -85,B 0,C 180,E1 -11386.718,E2 -11386.718} C_VEL
LIN {X 0,Y 395.975,Z 277.731,A -85,B 0,C 180,E1 -11388.196,E2 -11388.196} C_VEL
LIN {X 0,Y 396.172,Z 275.274,A -85,B 0,C 180,E1 -11389.712,E2 -11389.712} C_VEL
LIN {X 0,Y 396.481,Z 270.665,A -85,B 0,C 180,E1 -11391.654,E2 -11391.654} C_VEL
LIN {X 0,Y 396.889,Z 265.364,A -85,B 0,C 180,E1 -11393.299,E2 -11393.299} C_VEL
LIN {X 0,Y 397.33,Z 259.507,A -85,B 0,C 180,E1 -11394.739,E2 -11394.739} C_VEL
LIN {X 0,Y 397.988,Z 251.631,A -85,B 0,C 180,E1 -11396.299,E2 -11396.299} C_VEL
LIN {X 0,Y 398.771,Z 242.272,A -85,B 0,C 180,E1 -11397.774,E2 -11397.774} C_VEL
LIN {X 0,Y 399.509,Z 232.429,A -85,B 0,C 180,E1 -11399.032,E2 -11399.032} C_VEL
LIN {X 0,Y 400.197,Z 221.969,A -85,B 0,C 180,E1 -11400.112,E2 -11400.112} C_VEL
LIN {X 0,Y 400.988,Z 209.763,A -85,B 0,C 180,E1 -11401.102,E2 -11401.102} C_VEL
LIN {X 0,Y 401.528,Z 198.761,A -85,B 0,C 180,E1 -11401.798,E2 -11401.798} C_VEL
LIN {X 0,Y 398.679,Z 186.004,A -85,B 0,C 180,E1 -11402.54,E2 -11402.54} C_VEL
LIN {X 0,Y 396.239,Z 176.232,A -85,B 0,C 180,E1 -11403.002,E2 -11403.002} C_VEL
LIN {X 0,Y 396.27,Z 173.166,A -85,B 0,C 180,E1 -11405.926,E2 -11405.926} C_VEL
LIN {X 0,Y 396.359,Z 168.953,A -85,B 0,C 180,E1 -11410.01,E2 -11410.01} C_VEL
LIN {X 0,Y 396.475,Z 165.405,A -85,B 0,C 180,E1 -11413.523,E2 -11413.523} C_VEL
LIN {X 0,Y 396.528,Z 163.31,A -85,B 0,C 180,E1 -11415.633,E2 -11415.633} C_VEL
LIN {X 0,Y 396.832,Z 163.055,A -85,B 0,C 180,E1 -11417.73,E2 -11417.73} C_VEL
LIN {X 0,Y 397.172,Z 163.011,A -85,B 0,C 180,E1 -11420.836,E2 -11420.836} C_VEL
LIN {X 0,Y 397.329,Z 162.991,A -85,B 0,C 180,E1 -11422.887,E2 -11422.887} C_VEL
LIN {X 0,Y 397.248,Z 163.001,A -85,B 0,C 180,E1 -11424.925,E2 -11424.925} C_VEL
LIN {X 0,Y 397.449,Z 162.979,A -85,B 0,C 180,E1 -11427.973,E2 -11427.973} C_VEL
LIN {X 0,Y 397.578,Z 162.964,A -85,B 0,C 180,E1 -11430,E2 -11430} C_VEL
LIN {X 0,Y 397.378,Z 162.984,A -85,B 0,C 180,E1 -11433.041,E2 -11433.041} C_VEL
LIN {X 0,Y 397.359,Z 162.987,A -85,B 0,C 180,E1 -11437.112,E2 -11437.112} C_VEL
LIN {X 0,Y 397.215,Z 163.008,A -85,B 0,C 180,E1 -11440.191,E2 -11440.191} C_VEL
LIN {X 0,Y 397.212,Z 163.006,A -85,B 0,C 180,E1 -11442.207,E2 -11442.207} C_VEL
LIN {X 0,Y 396.581,Z 163.088,A -85,B 0,C 180,E1 -11443.053,E2 -11443.053} C_VEL
LIN {X 0,Y 393.691,Z 163.447,A -85,B 0,C 180,E1 -11444.426,E2 -11444.426} C_VEL
LIN {X 0,Y 391.232,Z 163.754,A -85,B 0,C 180,E1 -11445.536,E2 -11445.536} C_VEL
LIN {X 0,Y 390.2,Z 163.879,A -85,B 0,C 180,E1 -11446.396,E2 -11446.396} C_VEL
LIN {X 0,Y 390.131,Z 163.887,A -85,B 0,C 180,E1 -11446.687,E2 -11446.687} C_VEL
LIN {X 0,Y 390.1,Z 163.893,A -85,B 0,C 180,E1 -11450.017,E2 -11450.017} C_VEL
LIN {X 0,Y 390.086,Z 163.897,A -85,B 0,C 180,E1 -11453.351,E2 -11453.351} C_VEL
LIN {X 0,Y 390.11,Z 163.891,A -85,B 0,C 180,E1 -11456.768,E2 -11456.768} C_VEL
LIN {X 0,Y 390.036,Z 163.899,A -85,B 0,C 180,E1 -11460.3,E2 -11460.3} C_VEL
LIN {X 0,Y 390.065,Z 163.895,A -85,B 0,C 180,E1 -11464.025,E2 -11464.025} C_VEL
LIN {X 0,Y 390.04,Z 163.901,A -85,B 0,C 180,E1 -11467.551,E2 -11467.551} C_VEL
LIN {X 0,Y 390.054,Z 163.899,A -85,B 0,C 180,E1 -11470.822,E2 -11470.822} C_VEL
LIN {X 0,Y 390.054,Z 163.896,A -85,B 0,C 180,E1 -11473.887,E2 -11473.887} C_VEL
LIN {X 0,Y 390.055,Z 163.9,A -85,B 0,C 180,E1 -11476.79,E2 -11476.79} C_VEL
LIN {X 0,Y 390.054,Z 163.897,A -85,B 0,C 180,E1 -11479.561,E2 -11479.561} C_VEL
LIN {X 0,Y 390.044,Z 163.9,A -85,B 0,C 180,E1 -11482.449,E2 -11482.449} C_VEL
LIN {X 0,Y 390.066,Z 163.896,A -85,B 0,C 180,E1 -11486.046,E2 -11486.046} C_VEL
LIN {X 0,Y 390.045,Z 163.897,A -85,B 0,C 180,E1 -11489.87,E2 -11489.87} C_VEL
LIN {X 0,Y 390.112,Z 163.89,A -85,B 0,C 180,E1 -11493.232,E2 -11493.232} C_VEL
LIN {X 0,Y 390.106,Z 163.894,A -85,B 0,C 180,E1 -11496.751,E2 -11496.751} C_VEL
LIN {X 0,Y 390.103,Z 163.892,A -85,B 0,C 180,E1 -11499.984,E2 -11499.984} C_VEL
LIN {X 0,Y 390.138,Z 163.886,A -85,B 0,C 180,E1 -11503.249,E2 -11503.249} C_VEL
LIN {X 0,Y 390.195,Z 163.883,A -85,B 0,C 180,E1 -11506.562,E2 -11506.562} C_VEL
LIN {X 0,Y 390.169,Z 163.883,A -85,B 0,C 180,E1 -11509.623,E2 -11509.623} C_VEL
LIN {X 0,Y 390.296,Z 163.868,A -85,B 0,C 180,E1 -11512.759,E2 -11512.759} C_VEL
LIN {X 0,Y 390.227,Z 163.875,A -85,B 0,C 180,E1 -11514.834,E2 -11514.834} C_VEL
LIN {X 0,Y 390.422,Z 163.854,A -85,B 0,C 180,E1 -11517.937,E2 -11517.937} C_VEL
LIN {X 0,Y 390.55,Z 163.839,A -85,B 0,C 180,E1 -11520.001,E2 -11520.001} C_VEL
LIN {X 0,Y 390.311,Z 163.865,A -85,B 0,C 180,E1 -11523.097,E2 -11523.097} C_VEL
LIN {X 0,Y 390.301,Z 163.869,A -85,B 0,C 180,E1 -11526.203,E2 -11526.203} C_VEL
LIN {X 0,Y 390.195,Z 163.881,A -85,B 0,C 180,E1 -11529.33,E2 -11529.33} C_VEL
LIN {X 0,Y 390.173,Z 163.883,A -85,B 0,C 180,E1 -11532.484,E2 -11532.484} C_VEL
LIN {X 0,Y 390.141,Z 163.89,A -85,B 0,C 180,E1 -11535.677,E2 -11535.677} C_VEL
LIN {X 0,Y 390.108,Z 163.891,A -85,B 0,C 180,E1 -11538.922,E2 -11538.922} C_VEL
LIN {X 0,Y 390.042,Z 163.899,A -85,B 0,C 180,E1 -11542.235,E2 -11542.235} C_VEL
LIN {X 0,Y 390.122,Z 163.891,A -85,B 0,C 180,E1 -11545.744,E2 -11545.744} C_VEL
LIN {X 0,Y 390.061,Z 163.899,A -85,B 0,C 180,E1 -11549.11,E2 -11549.11} C_VEL
LIN {X 0,Y 390.045,Z 163.899,A -85,B 0,C 180,E1 -11552.722,E2 -11552.722} C_VEL
LIN {X 0,Y 390.058,Z 163.897,A -85,B 0,C 180,E1 -11555.826,E2 -11555.826} C_VEL
LIN {X 0,Y 390.071,Z 163.899,A -85,B 0,C 180,E1 -11559.218,E2 -11559.218} C_VEL
LIN {X 0,Y 390.045,Z 163.897,A -85,B 0,C 180,E1 -11562.374,E2 -11562.374} C_VEL
LIN {X 0,Y 390.089,Z 163.996,A -85,B 0,C 180,E1 -11565.361,E2 -11565.361} C_VEL
LIN {X 0,Y 391.246,Z 170.329,A -85,B 0,C 180,E1 -11568.978,E2 -11568.978} C_VEL
LIN {X 0,Y 392.257,Z 175.985,A -85,B 0,C 180,E1 -11572.031,E2 -11572.031} C_VEL
LIN {X 0,Y 392.506,Z 179.433,A -85,B 0,C 180,E1 -11573.781,E2 -11573.781} C_VEL
LIN {X 0,Y 392.111,Z 184.569,A -85,B 0,C 180,E1 -11576.246,E2 -11576.246} C_VEL
LIN {X 0,Y 391.673,Z 189.699,A -85,B 0,C 180,E1 -11578.644,E2 -11578.644} C_VEL
LIN {X 0,Y 390.985,Z 197.444,A -85,B 0,C 180,E1 -11582.138,E2 -11582.138} C_VEL
LIN {X 0,Y 390.371,Z 205.197,A -85,B 0,C 180,E1 -11585.539,E2 -11585.539} C_VEL
LIN {X 0,Y 389.918,Z 212.975,A -85,B 0,C 180,E1 -11588.87,E2 -11588.87} C_VEL
LIN {X 0,Y 389.575,Z 219.078,A -85,B 0,C 180,E1 -11591.427,E2 -11591.427} C_VEL
LIN {X 0,Y 392.164,Z 234.896,A -85,B 0,C 180,E1 -11592.106,E2 -11592.106} C_VEL
LIN {X 0,Y 393.843,Z 247.738,A -85,B 0,C 180,E1 -11592.849,E2 -11592.849} C_VEL
LIN {X 0,Y 394.08,Z 252.929,A -85,B 0,C 180,E1 -11593.196,E2 -11593.196} C_VEL
LIN {X 0,Y 393.181,Z 264.262,A -85,B 0,C 180,E1 -11594.049,E2 -11594.049} C_VEL
LIN {X 0,Y 392.307,Z 274.988,A -85,B 0,C 180,E1 -11595.077,E2 -11595.077} C_VEL
LIN {X 0,Y 391.54,Z 285.05,A -85,B 0,C 180,E1 -11596.277,E2 -11596.277} C_VEL
LIN {X 0,Y 390.778,Z 293.721,A -85,B 0,C 180,E1 -11597.537,E2 -11597.537} C_VEL
LIN {X 0,Y 389.971,Z 302.449,A -85,B 0,C 180,E1 -11599.092,E2 -11599.092} C_VEL
LIN {X 0,Y 389.454,Z 309.423,A -85,B 0,C 180,E1 -11600.653,E2 -11600.653} C_VEL
LIN {X 0,Y 389.077,Z 315.013,A -85,B 0,C 180,E1 -11602.214,E2 -11602.214} C_VEL
LIN {X 0,Y 388.83,Z 320.191,A -85,B 0,C 180,E1 -11604.102,E2 -11604.102} C_VEL
LIN {X 0,Y 388.727,Z 323.605,A -85,B 0,C 180,E1 -11605.853,E2 -11605.853} C_VEL
LIN {X 0,Y 388.704,Z 325.018,A -85,B 0,C 180,E1 -11606.891,E2 -11606.891} C_VEL
LIN {X 0,Y 388.787,Z 326.024,A -85,B 0,C 180,E1 -11607.928,E2 -11607.928} C_VEL
LIN {X 0,Y 388.733,Z 326.837,A -85,B 0,C 180,E1 -11610,E2 -11610} C_VEL
LIN {X 0,Y 388.735,Z 326.607,A -85,B 0,C 180,E1 -11611.036,E2 -11611.036} C_VEL
LIN {X 0,Y 388.77,Z 325.977,A -85,B 0,C 180,E1 -11612.072,E2 -11612.072} C_VEL
LIN {X 0,Y 388.73,Z 323.514,A -85,B 0,C 180,E1 -11614.147,E2 -11614.147} C_VEL
LIN {X 0,Y 388.831,Z 320.06,A -85,B 0,C 180,E1 -11615.9,E2 -11615.9} C_VEL
LIN {X 0,Y 389.079,Z 314.845,A -85,B 0,C 180,E1 -11617.786,E2 -11617.786} C_VEL
LIN {X 0,Y 389.451,Z 309.233,A -85,B 0,C 180,E1 -11619.347,E2 -11619.347} C_VEL
LIN {X 0,Y 389.961,Z 302.245,A -85,B 0,C 180,E1 -11620.908,E2 -11620.908} C_VEL
LIN {X 0,Y 390.78,Z 293.535,A -85,B 0,C 180,E1 -11622.464,E2 -11622.464} C_VEL
LIN {X 0,Y 391.661,Z 283.398,A -85,B 0,C 180,E1 -11623.92,E2 -11623.92} C_VEL
LIN {X 0,Y 392.385,Z 273.706,A -85,B 0,C 180,E1 -11625.053,E2 -11625.053} C_VEL
LIN {X 0,Y 393.309,Z 262.77,A -85,B 0,C 180,E1 -11626.08,E2 -11626.08} C_VEL
LIN {X 0,Y 394.201,Z 251.377,A -85,B 0,C 180,E1 -11626.922,E2 -11626.922} C_VEL
LIN {X 0,Y 392.803,Z 239.23,A -85,B 0,C 180,E1 -11627.708,E2 -11627.708} C_VEL
LIN {X 0,Y 390.986,Z 226.263,A -85,B 0,C 180,E1 -11628.354,E2 -11628.354} C_VEL
LIN {X 0,Y 389.557,Z 218.097,A -85,B 0,C 180,E1 -11628.677,E2 -11628.677} C_VEL
LIN {X 0,Y 389.889,Z 210.914,A -85,B 0,C 180,E1 -11631.687,E2 -11631.687} C_VEL
LIN {X 0,Y 390.396,Z 203.132,A -85,B 0,C 180,E1 -11635.028,E2 -11635.028} C_VEL
LIN {X 0,Y 390.954,Z 195.861,A -85,B 0,C 180,E1 -11638.254,E2 -11638.254} C_VEL
LIN {X 0,Y 391.726,Z 187.872,A -85,B 0,C 180,E1 -11641.947,E2 -11641.947} C_VEL
LIN {X 0,Y 392.482,Z 180.538,A -85,B 0,C 180,E1 -11645.589,E2 -11645.589} C_VEL
LIN {X 0,Y 392.38,Z 176.944,A -85,B 0,C 180,E1 -11647.516,E2 -11647.516} C_VEL
LIN {X 0,Y 391.391,Z 171.014,A -85,B 0,C 180,E1 -11651.046,E2 -11651.046} C_VEL
LIN {X 0,Y 390.364,Z 165.679,A -85,B 0,C 180,E1 -11654.6,E2 -11654.6} C_VEL
LIN {X 0,Y 390.059,Z 163.901,A -85,B 0,C 180,E1 -11655.989,E2 -11655.989} C_VEL
LIN {X 0,Y 390.061,Z 163.902,A -85,B 0,C 180,E1 -11659.561,E2 -11659.561} C_VEL
LIN {X 0,Y 390.048,Z 163.901,A -85,B 0,C 180,E1 -11662.449,E2 -11662.449} C_VEL
LIN {X 0,Y 390.072,Z 163.897,A -85,B 0,C 180,E1 -11666.045,E2 -11666.045} C_VEL
LIN {X 0,Y 390.051,Z 163.9,A -85,B 0,C 180,E1 -11669.869,E2 -11669.869} C_VEL
LIN {X 0,Y 390.118,Z 163.89,A -85,B 0,C 180,E1 -11673.232,E2 -11673.232} C_VEL
LIN {X 0,Y 390.111,Z 163.893,A -85,B 0,C 180,E1 -11676.75,E2 -11676.75} C_VEL
LIN {X 0,Y 390.108,Z 163.891,A -85,B 0,C 180,E1 -11679.983,E2 -11679.983} C_VEL
LIN {X 0,Y 390.142,Z 163.889,A -85,B 0,C 180,E1 -11683.248,E2 -11683.248} C_VEL
LIN {X 0,Y 390.199,Z 163.883,A -85,B 0,C 180,E1 -11686.561,E2 -11686.561} C_VEL
LIN {X 0,Y 390.209,Z 163.881,A -85,B 0,C 180,E1 -11690.671,E2 -11690.671} C_VEL
LIN {X 0,Y 390.323,Z 163.867,A -85,B 0,C 180,E1 -11692.759,E2 -11692.759} C_VEL
LIN {X 0,Y 390.231,Z 163.878,A -85,B 0,C 180,E1 -11694.833,E2 -11694.833} C_VEL
LIN {X 0,Y 390.425,Z 163.853,A -85,B 0,C 180,E1 -11697.936,E2 -11697.936} C_VEL
LIN {X 0,Y 390.554,Z 163.839,A -85,B 0,C 180,E1 -11699.999,E2 -11699.999} C_VEL
LIN {X 0,Y 390.318,Z 163.868,A -85,B 0,C 180,E1 -11703.096,E2 -11703.096} C_VEL
LIN {X 0,Y 390.299,Z 163.871,A -85,B 0,C 180,E1 -11706.608,E2 -11706.608} C_VEL
LIN {X 0,Y 390.105,Z 163.895,A -85,B 0,C 180,E1 -11709.331,E2 -11709.331} C_VEL
LIN {X 0,Y 390.03,Z 164.09,A -85,B 0,C 180,E1 -11710.38,E2 -11710.38} C_VEL
LIN {X 0,Y 389.947,Z 166.845,A -85,B 0,C 180,E1 -11713.55,E2 -11713.55} C_VEL
LIN {X 0,Y 389.734,Z 169.989,A -85,B 0,C 180,E1 -11717.109,E2 -11717.109} C_VEL
LIN {X 0,Y 389.561,Z 172.861,A -85,B 0,C 180,E1 -11720.26,E2 -11720.26} C_VEL
LIN {X 0,Y 389.448,Z 175.767,A -85,B 0,C 180,E1 -11723.391,E2 -11723.391} C_VEL
LIN {X 0,Y 389.389,Z 178.838,A -85,B 0,C 180,E1 -11726.424,E2 -11726.424} C_VEL
LIN {X 0,Y 393.242,Z 191.949,A -85,B 0,C 180,E1 -11727.147,E2 -11727.147} C_VEL
LIN {X 0,Y 395.427,Z 201.976,A -85,B 0,C 180,E1 -11727.81,E2 -11727.81} C_VEL
LIN {X 0,Y 394.726,Z 213.543,A -85,B 0,C 180,E1 -11728.587,E2 -11728.587} C_VEL
LIN {X 0,Y 393.922,Z 224.339,A -85,B 0,C 180,E1 -11729.513,E2 -11729.513} C_VEL
LIN {X 0,Y 393.199,Z 234.169,A -85,B 0,C 180,E1 -11730.571,E2 -11730.571} C_VEL
LIN {X 0,Y 392.273,Z 244.226,A -85,B 0,C 180,E1 -11731.905,E2 -11731.905} C_VEL
LIN {X 0,Y 391.532,Z 252.14,A -85,B 0,C 180,E1 -11733.193,E2 -11733.193} C_VEL
LIN {X 0,Y 390.714,Z 259.48,A -85,B 0,C 180,E1 -11734.645,E2 -11734.645} C_VEL
LIN {X 0,Y 390.19,Z 265.518,A -85,B 0,C 180,E1 -11736.129,E2 -11736.129} C_VEL
LIN {X 0,Y 389.698,Z 270.927,A -85,B 0,C 180,E1 -11737.818,E2 -11737.818} C_VEL
LIN {X 0,Y 389.369,Z 274.325,A -85,B 0,C 180,E1 -11739.178,E2 -11739.178} C_VEL
LIN {X 0,Y 389.097,Z 277.095,A -85,B 0,C 180,E1 -11740.657,E2 -11740.657} C_VEL
LIN {X 0,Y 388.855,Z 279.04,A -85,B 0,C 180,E1 -11742.181,E2 -11742.181} C_VEL
LIN {X 0,Y 388.716,Z 280.09,A -85,B 0,C 180,E1 -11743.68,E2 -11743.68} C_VEL
LIN {X 0,Y 388.673,Z 280.314,A -85,B 0,C 180,E1 -11745.154,E2 -11745.154} C_VEL
LIN {X 0,Y 388.715,Z 279.753,A -85,B 0,C 180,E1 -11746.603,E2 -11746.603} C_VEL
LIN {X 0,Y 388.884,Z 278.387,A -85,B 0,C 180,E1 -11748.035,E2 -11748.035} C_VEL
LIN {X 0,Y 389.056,Z 276.299,A -85,B 0,C 180,E1 -11749.434,E2 -11749.434} C_VEL
LIN {X 0,Y 389.271,Z 273.213,A -85,B 0,C 180,E1 -11750.925,E2 -11750.925} C_VEL
LIN {X 0,Y 389.63,Z 268.792,A -85,B 0,C 180,E1 -11752.527,E2 -11752.527} C_VEL
LIN {X 0,Y 390.112,Z 262.978,A -85,B 0,C 180,E1 -11754.162,E2 -11754.162} C_VEL
LIN {X 0,Y 390.709,Z 255.448,A -85,B 0,C 180,E1 -11755.835,E2 -11755.835} C_VEL
LIN {X 0,Y 391.552,Z 246.381,A -85,B 0,C 180,E1 -11757.42,E2 -11757.42} C_VEL
LIN {X 0,Y 392.255,Z 237.417,A -85,B 0,C 180,E1 -11758.695,E2 -11758.695} C_VEL
LIN {X 0,Y 393.06,Z 226.411,A -85,B 0,C 180,E1 -11759.957,E2 -11759.957} C_VEL
LIN {X 0,Y 393.797,Z 215.142,A -85,B 0,C 180,E1 -11760.983,E2 -11760.983} C_VEL
LIN {X 0,Y 394.581,Z 203.177,A -85,B 0,C 180,E1 -11761.833,E2 -11761.833} C_VEL
LIN {X 0,Y 394.632,Z 199.902,A -85,B 0,C 180,E1 -11762.029,E2 -11762.029} C_VEL
LIN {X 0,Y 391.765,Z 186.921,A -85,B 0,C 180,E1 -11762.813,E2 -11762.813} C_VEL
LIN {X 0,Y 389.175,Z 176.625,A -85,B 0,C 180,E1 -11763.307,E2 -11763.307} C_VEL
LIN {X 0,Y 389.183,Z 173.21,A -85,B 0,C 180,E1 -11766.591,E2 -11766.591} C_VEL
LIN {X 0,Y 389.306,Z 169.801,A -85,B 0,C 180,E1 -11769.94,E2 -11769.94} C_VEL
LIN {X 0,Y 389.411,Z 166.516,A -85,B 0,C 180,E1 -11773.216,E2 -11773.216} C_VEL
LIN {X 0,Y 389.458,Z 164.397,A -85,B 0,C 180,E1 -11775.366,E2 -11775.366} C_VEL
LIN {X 0,Y 389.664,Z 163.948,A -85,B 0,C 180,E1 -11776.89,E2 -11776.89} C_VEL
LIN {X 0,Y 390.02,Z 163.902,A -85,B 0,C 180,E1 -11779.619,E2 -11779.619} C_VEL
LIN {X 0,Y 390.278,Z 163.87,A -85,B 0,C 180,E1 -11782.758,E2 -11782.758} C_VEL
LIN {X 0,Y 390.22,Z 163.877,A -85,B 0,C 180,E1 -11784.833,E2 -11784.833} C_VEL
LIN {X 0,Y 390.418,Z 163.855,A -85,B 0,C 180,E1 -11787.937,E2 -11787.937} C_VEL
LIN {X 0,Y 390.547,Z 163.84,A -85,B 0,C 180,E1 -11790,E2 -11790} C_VEL
LIN {X 0,Y 390.312,Z 163.864,A -85,B 0,C 180,E1 -11793.096,E2 -11793.096} C_VEL
LIN {X 0,Y 390.324,Z 163.866,A -85,B 0,C 180,E1 -11796.202,E2 -11796.202} C_VEL
LIN {X 0,Y 390.311,Z 163.867,A -85,B 0,C 180,E1 -11798.282,E2 -11798.282} C_VEL
LIN {X 0,Y 390.167,Z 163.883,A -85,B 0,C 180,E1 -11802.483,E2 -11802.483} C_VEL
LIN {X 0,Y 390.136,Z 163.891,A -85,B 0,C 180,E1 -11805.677,E2 -11805.677} C_VEL
LIN {X 0,Y 390.131,Z 163.887,A -85,B 0,C 180,E1 -11806.687,E2 -11806.687} C_VEL
LIN {X 0,Y 389.494,Z 163.97,A -85,B 0,C 180,E1 -11807.548,E2 -11807.548} C_VEL
LIN {X 0,Y 386.614,Z 164.325,A -85,B 0,C 180,E1 -11808.947,E2 -11808.947} C_VEL
LIN {X 0,Y 384.147,Z 164.634,A -85,B 0,C 180,E1 -11810.078,E2 -11810.078} C_VEL
LIN {X 0,Y 383.08,Z 164.766,A -85,B 0,C 180,E1 -11810.954,E2 -11810.954} C_VEL
LIN {X 0,Y 382.991,Z 164.778,A -85,B 0,C 180,E1 -11811.25,E2 -11811.25} C_VEL
LIN {X 0,Y 383.03,Z 164.775,A -85,B 0,C 180,E1 -11813.807,E2 -11813.807} C_VEL
LIN {X 0,Y 383.076,Z 164.766,A -85,B 0,C 180,E1 -11816.123,E2 -11816.123} C_VEL
LIN {X 0,Y 382.989,Z 164.78,A -85,B 0,C 180,E1 -11819.7,E2 -11819.7} C_VEL
LIN {X 0,Y 383,Z 164.78,A -85,B 0,C 180,E1 -11823.401,E2 -11823.401} C_VEL
LIN {X 0,Y 383.029,Z 164.772,A -85,B 0,C 180,E1 -11826.165,E2 -11826.165} C_VEL
LIN {X 0,Y 383.006,Z 164.775,A -85,B 0,C 180,E1 -11829.959,E2 -11829.959} C_VEL
LIN {X 0,Y 383.002,Z 164.778,A -85,B 0,C 180,E1 -11832.779,E2 -11832.779} C_VEL
LIN {X 0,Y 382.995,Z 164.776,A -85,B 0,C 180,E1 -11835.79,E2 -11835.79} C_VEL
LIN {X 0,Y 382.986,Z 164.781,A -85,B 0,C 180,E1 -11838.796,E2 -11838.796} C_VEL
LIN {X 0,Y 382.999,Z 164.776,A -85,B 0,C 180,E1 -11842.096,E2 -11842.096} C_VEL
LIN {X 0,Y 383.016,Z 164.775,A -85,B 0,C 180,E1 -11845.333,E2 -11845.333} C_VEL
LIN {X 0,Y 382.981,Z 164.78,A -85,B 0,C 180,E1 -11849.082,E2 -11849.082} C_VEL
LIN {X 0,Y 383.056,Z 164.773,A -85,B 0,C 180,E1 -11852.699,E2 -11852.699} C_VEL
LIN {X 0,Y 383.051,Z 164.771,A -85,B 0,C 180,E1 -11855.04,E2 -11855.04} C_VEL
LIN {X 0,Y 382.999,Z 164.779,A -85,B 0,C 180,E1 -11858.47,E2 -11858.47} C_VEL
LIN {X 0,Y 383.062,Z 164.768,A -85,B 0,C 180,E1 -11861.827,E2 -11861.827} C_VEL
LIN {X 0,Y 383.11,Z 164.761,A -85,B 0,C 180,E1 -11865.119,E2 -11865.119} C_VEL
LIN {X 0,Y 383.099,Z 164.768,A -85,B 0,C 180,E1 -11868.359,E2 -11868.359} C_VEL
LIN {X 0,Y 383.262,Z 164.746,A -85,B 0,C 180,E1 -11871.978,E2 -11871.978} C_VEL
LIN {X 0,Y 383.198,Z 164.751,A -85,B 0,C 180,E1 -11874.739,E2 -11874.739} C_VEL
LIN {X 0,Y 383.389,Z 164.73,A -85,B 0,C 180,E1 -11877.899,E2 -11877.899} C_VEL
LIN {X 0,Y 383.519,Z 164.715,A -85,B 0,C 180,E1 -11880.001,E2 -11880.001} C_VEL
LIN {X 0,Y 383.248,Z 164.745,A -85,B 0,C 180,E1 -11883.154,E2 -11883.154} C_VEL
LIN {X 0,Y 383.258,Z 164.745,A -85,B 0,C 180,E1 -11886.317,E2 -11886.317} C_VEL
LIN {X 0,Y 383.145,Z 164.76,A -85,B 0,C 180,E1 -11889.503,E2 -11889.503} C_VEL
LIN {X 0,Y 383.138,Z 164.758,A -85,B 0,C 180,E1 -11892.717,E2 -11892.717} C_VEL
LIN {X 0,Y 383.083,Z 164.768,A -85,B 0,C 180,E1 -11895.974,E2 -11895.974} C_VEL
LIN {X 0,Y 383.063,Z 164.77,A -85,B 0,C 180,E1 -11899.284,E2 -11899.284} C_VEL
LIN {X 0,Y 383.04,Z 164.775,A -85,B 0,C 180,E1 -11903.451,E2 -11903.451} C_VEL
LIN {X 0,Y 383.082,Z 164.765,A -85,B 0,C 180,E1 -11906.124,E2 -11906.124} C_VEL
LIN {X 0,Y 382.994,Z 164.779,A -85,B 0,C 180,E1 -11909.7,E2 -11909.7} C_VEL
LIN {X 0,Y 383.005,Z 164.779,A -85,B 0,C 180,E1 -11913.401,E2 -11913.401} C_VEL
LIN {X 0,Y 383.034,Z 164.771,A -85,B 0,C 180,E1 -11916.165,E2 -11916.165} C_VEL
LIN {X 0,Y 383.01,Z 164.777,A -85,B 0,C 180,E1 -11919.959,E2 -11919.959} C_VEL
LIN {X 0,Y 383.007,Z 164.774,A -85,B 0,C 180,E1 -11922.779,E2 -11922.779} C_VEL
LIN {X 0,Y 383.023,Z 164.789,A -85,B 0,C 180,E1 -11924.949,E2 -11924.949} C_VEL
LIN {X 0,Y 384.157,Z 171.027,A -85,B 0,C 180,E1 -11928.598,E2 -11928.598} C_VEL
LIN {X 0,Y 385.177,Z 176.608,A -85,B 0,C 180,E1 -11931.683,E2 -11931.683} C_VEL
LIN {X 0,Y 385.52,Z 179.778,A -85,B 0,C 180,E1 -11933.334,E2 -11933.334} C_VEL
LIN {X 0,Y 385.206,Z 184.269,A -85,B 0,C 180,E1 -11935.557,E2 -11935.557} C_VEL
LIN {X 0,Y 384.653,Z 190.682,A -85,B 0,C 180,E1 -11938.619,E2 -11938.619} C_VEL
LIN {X 0,Y 383.936,Z 198.387,A -85,B 0,C 180,E1 -11942.175,E2 -11942.175} C_VEL
LIN {X 0,Y 383.289,Z 206.152,A -85,B 0,C 180,E1 -11945.634,E2 -11945.634} C_VEL
LIN {X 0,Y 382.817,Z 213.883,A -85,B 0,C 180,E1 -11949.024,E2 -11949.024} C_VEL
LIN {X 0,Y 382.549,Z 218.861,A -85,B 0,C 180,E1 -11951.123,E2 -11951.123} C_VEL
LIN {X 0,Y 384.83,Z 232.315,A -85,B 0,C 180,E1 -11951.673,E2 -11951.673} C_VEL
LIN {X 0,Y 386.545,Z 245.894,A -85,B 0,C 180,E1 -11952.444,E2 -11952.444} C_VEL
LIN {X 0,Y 387.234,Z 252.525,A -85,B 0,C 180,E1 -11952.905,E2 -11952.905} C_VEL
LIN {X 0,Y 386.318,Z 263.685,A -85,B 0,C 180,E1 -11953.757,E2 -11953.757} C_VEL
LIN {X 0,Y 385.406,Z 274.45,A -85,B 0,C 180,E1 -11954.803,E2 -11954.803} C_VEL
LIN {X 0,Y 384.586,Z 284.739,A -85,B 0,C 180,E1 -11956.052,E2 -11956.052} C_VEL
LIN {X 0,Y 383.64,Z 294.84,A -85,B 0,C 180,E1 -11957.57,E2 -11957.57} C_VEL
LIN {X 0,Y 382.848,Z 303.215,A -85,B 0,C 180,E1 -11959.155,E2 -11959.155} C_VEL
LIN {X 0,Y 382.335,Z 309.975,A -85,B 0,C 180,E1 -11960.744,E2 -11960.744} C_VEL
LIN {X 0,Y 381.927,Z 316.179,A -85,B 0,C 180,E1 -11962.599,E2 -11962.599} C_VEL
LIN {X 0,Y 381.731,Z 320.12,A -85,B 0,C 180,E1 -11964.151,E2 -11964.151} C_VEL
LIN {X 0,Y 381.656,Z 323.172,A -85,B 0,C 180,E1 -11965.776,E2 -11965.776} C_VEL
LIN {X 0,Y 381.61,Z 324.59,A -85,B 0,C 180,E1 -11966.833,E2 -11966.833} C_VEL
LIN {X 0,Y 381.702,Z 325.599,A -85,B 0,C 180,E1 -11967.89,E2 -11967.89} C_VEL
LIN {X 0,Y 381.668,Z 326.205,A -85,B 0,C 180,E1 -11968.945,E2 -11968.945} C_VEL
LIN {X 0,Y 381.663,Z 326.418,A -85,B 0,C 180,E1 -11970,E2 -11970} C_VEL
LIN {X 0,Y 381.668,Z 326.192,A -85,B 0,C 180,E1 -11971.055,E2 -11971.055} C_VEL
LIN {X 0,Y 381.688,Z 325.562,A -85,B 0,C 180,E1 -11972.111,E2 -11972.111} C_VEL
LIN {X 0,Y 381.658,Z 323.102,A -85,B 0,C 180,E1 -11974.224,E2 -11974.224} C_VEL
LIN {X 0,Y 381.732,Z 320.019,A -85,B 0,C 180,E1 -11975.851,E2 -11975.851} C_VEL
LIN {X 0,Y 381.929,Z 316.057,A -85,B 0,C 180,E1 -11977.401,E2 -11977.401} C_VEL
LIN {X 0,Y 382.334,Z 309.859,A -85,B 0,C 180,E1 -11979.256,E2 -11979.256} C_VEL
LIN {X 0,Y 382.838,Z 303.105,A -85,B 0,C 180,E1 -11980.846,E2 -11980.846} C_VEL
LIN {X 0,Y 383.634,Z 294.758,A -85,B 0,C 180,E1 -11982.431,E2 -11982.431} C_VEL
LIN {X 0,Y 384.429,Z 286.236,A -85,B 0,C 180,E1 -11983.749,E2 -11983.749} C_VEL
LIN {X 0,Y 385.288,Z 275.747,A -85,B 0,C 180,E1 -11985.066,E2 -11985.066} C_VEL
LIN {X 0,Y 386.35,Z 264.011,A -85,B 0,C 180,E1 -11986.242,E2 -11986.242} C_VEL
LIN {X 0,Y 387.294,Z 252.994,A -85,B 0,C 180,E1 -11987.107,E2 -11987.107} C_VEL
LIN {X 0,Y 386.484,Z 244.47,A -85,B 0,C 180,E1 -11987.708,E2 -11987.708} C_VEL
LIN {X 0,Y 384.91,Z 231.495,A -85,B 0,C 180,E1 -11988.456,E2 -11988.456} C_VEL
LIN {X 0,Y 382.545,Z 217.635,A -85,B 0,C 180,E1 -11989.067,E2 -11989.067} C_VEL
LIN {X 0,Y 382.865,Z 210.554,A -85,B 0,C 180,E1 -11992.105,E2 -11992.105} C_VEL
LIN {X 0,Y 383.415,Z 202.826,A -85,B 0,C 180,E1 -11995.516,E2 -11995.516} C_VEL
LIN {X 0,Y 384.072,Z 195.205,A -85,B 0,C 180,E1 -11999.007,E2 -11999.007} C_VEL
LIN {X 0,Y 384.876,Z 187.191,A -85,B 0,C 180,E1 -12002.861,E2 -12002.861} C_VEL
LIN {X 0,Y 385.51,Z 181.646,A -85,B 0,C 180,E1 -12005.688,E2 -12005.688} C_VEL
LIN {X 0,Y 385.405,Z 178.072,A -85,B 0,C 180,E1 -12007.645,E2 -12007.645} C_VEL
LIN {X 0,Y 384.332,Z 171.885,A -85,B 0,C 180,E1 -12011.432,E2 -12011.432} C_VEL
LIN {X 0,Y 383.51,Z 167.555,A -85,B 0,C 180,E1 -12014.381,E2 -12014.381} C_VEL
LIN {X 0,Y 383.02,Z 164.78,A -85,B 0,C 180,E1 -12016.521,E2 -12016.521} C_VEL
LIN {X 0,Y 383.02,Z 164.78,A -85,B 0,C 180,E1 -12020.413,E2 -12020.413} C_VEL
LIN {X 0,Y 383.029,Z 164.774,A -85,B 0,C 180,E1 -12024.044,E2 -12024.044} C_VEL
LIN {X 0,Y 382.991,Z 164.778,A -85,B 0,C 180,E1 -12027.578,E2 -12027.578} C_VEL
LIN {X 0,Y 382.997,Z 164.78,A -85,B 0,C 180,E1 -12030.3,E2 -12030.3} C_VEL
LIN {X 0,Y 383.061,Z 164.77,A -85,B 0,C 180,E1 -12032.698,E2 -12032.698} C_VEL
LIN {X 0,Y 383.057,Z 164.77,A -85,B 0,C 180,E1 -12035.04,E2 -12035.04} C_VEL
LIN {X 0,Y 382.998,Z 164.78,A -85,B 0,C 180,E1 -12038.469,E2 -12038.469} C_VEL
LIN {X 0,Y 383.057,Z 164.768,A -85,B 0,C 180,E1 -12041.826,E2 -12041.826} C_VEL
LIN {X 0,Y 383.114,Z 164.764,A -85,B 0,C 180,E1 -12045.118,E2 -12045.118} C_VEL
LIN {X 0,Y 383.102,Z 164.766,A -85,B 0,C 180,E1 -12048.358,E2 -12048.358} C_VEL
LIN {X 0,Y 383.308,Z 164.74,A -85,B 0,C 180,E1 -12051.932,E2 -12051.932} C_VEL
LIN {X 0,Y 383.204,Z 164.754,A -85,B 0,C 180,E1 -12054.738,E2 -12054.738} C_VEL
LIN {X 0,Y 383.392,Z 164.729,A -85,B 0,C 180,E1 -12057.898,E2 -12057.898} C_VEL
LIN {X 0,Y 383.524,Z 164.714,A -85,B 0,C 180,E1 -12059.999,E2 -12059.999} C_VEL
LIN {X 0,Y 383.254,Z 164.748,A -85,B 0,C 180,E1 -12063.153,E2 -12063.153} C_VEL
LIN {X 0,Y 383.259,Z 164.749,A -85,B 0,C 180,E1 -12066.598,E2 -12066.598} C_VEL
LIN {X 0,Y 383.061,Z 164.772,A -85,B 0,C 180,E1 -12069.504,E2 -12069.504} C_VEL
LIN {X 0,Y 382.96,Z 166.231,A -85,B 0,C 180,E1 -12071.646,E2 -12071.646} C_VEL
LIN {X 0,Y 382.884,Z 168.071,A -85,B 0,C 180,E1 -12073.805,E2 -12073.805} C_VEL
LIN {X 0,Y 382.687,Z 171.093,A -85,B 0,C 180,E1 -12077.258,E2 -12077.258} C_VEL
LIN {X 0,Y 382.522,Z 173.954,A -85,B 0,C 180,E1 -12080.443,E2 -12080.443} C_VEL
LIN {X 0,Y 382.353,Z 177.079,A -85,B 0,C 180,E1 -12083.852,E2 -12083.852} C_VEL
LIN {X 0,Y 382.329,Z 179.197,A -85,B 0,C 180,E1 -12086.03,E2 -12086.03} C_VEL
LIN {X 0,Y 386.379,Z 192.863,A -85,B 0,C 180,E1 -12086.809,E2 -12086.809} C_VEL
LIN {X 0,Y 388.697,Z 203.29,A -85,B 0,C 180,E1 -12087.528,E2 -12087.528} C_VEL
LIN {X 0,Y 387.946,Z 214.688,A -85,B 0,C 180,E1 -12088.32,E2 -12088.32} C_VEL
LIN {X 0,Y 387.028,Z 226.239,A -85,B 0,C 180,E1 -12089.359,E2 -12089.359} C_VEL
LIN {X 0,Y 386.117,Z 237.435,A -85,B 0,C 180,E1 -12090.64,E2 -12090.64} C_VEL
LIN {X 0,Y 385.229,Z 246.628,A -85,B 0,C 180,E1 -12091.942,E2 -12091.942} C_VEL
LIN {X 0,Y 384.46,Z 254.223,A -85,B 0,C 180,E1 -12093.257,E2 -12093.257} C_VEL
LIN {X 0,Y 383.553,Z 262.049,A -85,B 0,C 180,E1 -12094.931,E2 -12094.931} C_VEL
LIN {X 0,Y 382.98,Z 268.492,A -85,B 0,C 180,E1 -12096.689,E2 -12096.689} C_VEL
LIN {X 0,Y 382.388,Z 273.917,A -85,B 0,C 180,E1 -12098.674,E2 -12098.674} C_VEL
LIN {X 0,Y 382.111,Z 276.746,A -85,B 0,C 180,E1 -12100.07,E2 -12100.07} C_VEL
LIN {X 0,Y 381.895,Z 278.832,A -85,B 0,C 180,E1 -12101.49,E2 -12101.49} C_VEL
LIN {X 0,Y 381.676,Z 280.161,A -85,B 0,C 180,E1 -12102.944,E2 -12102.944} C_VEL
LIN {X 0,Y 381.607,Z 280.738,A -85,B 0,C 180,E1 -12104.413,E2 -12104.413} C_VEL
LIN {X 0,Y 381.605,Z 280.544,A -85,B 0,C 180,E1 -12105.91,E2 -12105.91} C_VEL
LIN {X 0,Y 381.7,Z 279.517,A -85,B 0,C 180,E1 -12107.433,E2 -12107.433} C_VEL
LIN {X 0,Y 381.899,Z 277.576,A -85,B 0,C 180,E1 -12108.982,E2 -12108.982} C_VEL
LIN {X 0,Y 382.155,Z 274.64,A -85,B 0,C 180,E1 -12110.569,E2 -12110.569} C_VEL
LIN {X 0,Y 382.474,Z 270.554,A -85,B 0,C 180,E1 -12112.196,E2 -12112.196} C_VEL
LIN {X 0,Y 382.985,Z 264.424,A -85,B 0,C 180,E1 -12114.04,E2 -12114.04} C_VEL
LIN {X 0,Y 383.643,Z 256.702,A -85,B 0,C 180,E1 -12115.836,E2 -12115.836} C_VEL
LIN {X 0,Y 384.359,Z 249.06,A -85,B 0,C 180,E1 -12117.256,E2 -12117.256} C_VEL
LIN {X 0,Y 385.092,Z 240.57,A -85,B 0,C 180,E1 -12118.55,E2 -12118.55} C_VEL
LIN {X 0,Y 385.852,Z 230.634,A -85,B 0,C 180,E1 -12119.79,E2 -12119.79} C_VEL
LIN {X 0,Y 386.678,Z 219.501,A -85,B 0,C 180,E1 -12120.909,E2 -12120.909} C_VEL
LIN {X 0,Y 387.465,Z 208.436,A -85,B 0,C 180,E1 -12121.788,E2 -12121.788} C_VEL
LIN {X 0,Y 387.863,Z 202.277,A -85,B 0,C 180,E1 -12122.187,E2 -12122.187} C_VEL
LIN {X 0,Y 386.099,Z 193.185,A -85,B 0,C 180,E1 -12122.784,E2 -12122.784} C_VEL
LIN {X 0,Y 383.084,Z 180.926,A -85,B 0,C 180,E1 -12123.437,E2 -12123.437} C_VEL
LIN {X 0,Y 382.095,Z 177.014,A -85,B 0,C 180,E1 -12123.62,E2 -12123.62} C_VEL
LIN {X 0,Y 382.136,Z 173.683,A -85,B 0,C 180,E1 -12126.861,E2 -12126.861} C_VEL
LIN {X 0,Y 382.224,Z 169.842,A -85,B 0,C 180,E1 -12130.672,E2 -12130.672} C_VEL
LIN {X 0,Y 382.361,Z 166.551,A -85,B 0,C 180,E1 -12133.996,E2 -12133.996} C_VEL
LIN {X 0,Y 382.394,Z 165.487,A -85,B 0,C 180,E1 -12135.09,E2 -12135.09} C_VEL
LIN {X 0,Y 382.507,Z 164.842,A -85,B 0,C 180,E1 -12136.181,E2 -12136.181} C_VEL
LIN {X 0,Y 382.951,Z 164.782,A -85,B 0,C 180,E1 -12139.425,E2 -12139.425} C_VEL
LIN {X 0,Y 383.228,Z 164.749,A -85,B 0,C 180,E1 -12142.624,E2 -12142.624} C_VEL
LIN {X 0,Y 383.191,Z 164.753,A -85,B 0,C 180,E1 -12144.738,E2 -12144.738} C_VEL
LIN {X 0,Y 383.385,Z 164.732,A -85,B 0,C 180,E1 -12147.899,E2 -12147.899} C_VEL
LIN {X 0,Y 383.516,Z 164.716,A -85,B 0,C 180,E1 -12150,E2 -12150} C_VEL
LIN {X 0,Y 383.248,Z 164.744,A -85,B 0,C 180,E1 -12153.153,E2 -12153.153} C_VEL
LIN {X 0,Y 383.282,Z 164.742,A -85,B 0,C 180,E1 -12156.316,E2 -12156.316} C_VEL
LIN {X 0,Y 383.257,Z 164.744,A -85,B 0,C 180,E1 -12158.436,E2 -12158.436} C_VEL
LIN {X 0,Y 383.095,Z 164.767,A -85,B 0,C 180,E1 -12161.642,E2 -12161.642} C_VEL
LIN {X 0,Y 383.107,Z 164.762,A -85,B 0,C 180,E1 -12164.882,E2 -12164.882} C_VEL
LIN {X 0,Y 383.059,Z 164.769,A -85,B 0,C 180,E1 -12168.174,E2 -12168.174} C_VEL
LIN {X 0,Y 382.991,Z 164.778,A -85,B 0,C 180,E1 -12171.25,E2 -12171.25} C_VEL
LIN {X 0,Y 382.317,Z 164.867,A -85,B 0,C 180,E1 -12172.129,E2 -12172.129} C_VEL
LIN {X 0,Y 379.467,Z 165.225,A -85,B 0,C 180,E1 -12173.558,E2 -12173.558} C_VEL
LIN {X 0,Y 377.078,Z 165.519,A -85,B 0,C 180,E1 -12174.713,E2 -12174.713} C_VEL
LIN {X 0,Y 376.082,Z 165.641,A -85,B 0,C 180,E1 -12175.606,E2 -12175.606} C_VEL
LIN {X 0,Y 376.016,Z 165.646,A -85,B 0,C 180,E1 -12175.908,E2 -12175.908} C_VEL
LIN {X 0,Y 375.958,Z 165.655,A -85,B 0,C 180,E1 -12179.08,E2 -12179.08} C_VEL
LIN {X 0,Y 375.946,Z 165.656,A -85,B 0,C 180,E1 -12182.829,E2 -12182.829} C_VEL
LIN {X 0,Y 375.954,Z 165.657,A -85,B 0,C 180,E1 -12185.416,E2 -12185.416} C_VEL
LIN {X 0,Y 375.971,Z 165.65,A -85,B 0,C 180,E1 -12188.271,E2 -12188.271} C_VEL
LIN {X 0,Y 375.932,Z 165.657,A -85,B 0,C 180,E1 -12191.601,E2 -12191.601} C_VEL
LIN {X 0,Y 375.951,Z 165.657,A -85,B 0,C 180,E1 -12195.265,E2 -12195.265} C_VEL
LIN {X 0,Y 375.938,Z 165.659,A -85,B 0,C 180,E1 -12199.133,E2 -12199.133} C_VEL
LIN {X 0,Y 375.964,Z 165.652,A -85,B 0,C 180,E1 -12201.912,E2 -12201.912} C_VEL
LIN {X 0,Y 375.978,Z 165.651,A -85,B 0,C 180,E1 -12205.333,E2 -12205.333} C_VEL
LIN {X 0,Y 375.956,Z 165.656,A -85,B 0,C 180,E1 -12208.439,E2 -12208.439} C_VEL
LIN {X 0,Y 375.982,Z 165.651,A -85,B 0,C 180,E1 -12212.141,E2 -12212.141} C_VEL
LIN {X 0,Y 376.006,Z 165.65,A -85,B 0,C 180,E1 -12214.54,E2 -12214.54} C_VEL
LIN {X 0,Y 375.967,Z 165.653,A -85,B 0,C 180,E1 -12218.047,E2 -12218.047} C_VEL
LIN {X 0,Y 376.008,Z 165.646,A -85,B 0,C 180,E1 -12221.474,E2 -12221.474} C_VEL
LIN {X 0,Y 376.058,Z 165.641,A -85,B 0,C 180,E1 -12224.833,E2 -12224.833} C_VEL
LIN {X 0,Y 376.051,Z 165.644,A -85,B 0,C 180,E1 -12228.137,E2 -12228.137} C_VEL
LIN {X 0,Y 376.217,Z 165.623,A -85,B 0,C 180,E1 -12231.922,E2 -12231.922} C_VEL
LIN {X 0,Y 376.17,Z 165.627,A -85,B 0,C 180,E1 -12234.64,E2 -12234.64} C_VEL
LIN {X 0,Y 376.355,Z 165.606,A -85,B 0,C 180,E1 -12237.86,E2 -12237.86} C_VEL
LIN {X 0,Y 376.489,Z 165.59,A -85,B 0,C 180,E1 -12240.001,E2 -12240.001} C_VEL
LIN {X 0,Y 376.186,Z 165.624,A -85,B 0,C 180,E1 -12243.213,E2 -12243.213} C_VEL
LIN {X 0,Y 376.215,Z 165.621,A -85,B 0,C 180,E1 -12246.436,E2 -12246.436} C_VEL
LIN {X 0,Y 376.115,Z 165.637,A -85,B 0,C 180,E1 -12249.682,E2 -12249.682} C_VEL
LIN {X 0,Y 376.091,Z 165.64,A -85,B 0,C 180,E1 -12253.658,E2 -12253.658} C_VEL
LIN {X 0,Y 376.046,Z 165.646,A -85,B 0,C 180,E1 -12257.608,E2 -12257.608} C_VEL
LIN {X 0,Y 375.98,Z 165.65,A -85,B 0,C 180,E1 -12260.833,E2 -12260.833} C_VEL
LIN {X 0,Y 375.996,Z 165.648,A -85,B 0,C 180,E1 -12264.282,E2 -12264.282} C_VEL
LIN {X 0,Y 376.022,Z 165.644,A -85,B 0,C 180,E1 -12266.652,E2 -12266.652} C_VEL
LIN {X 0,Y 375.967,Z 165.651,A -85,B 0,C 180,E1 -12270.313,E2 -12270.313} C_VEL
LIN {X 0,Y 375.962,Z 165.652,A -85,B 0,C 180,E1 -12274.112,E2 -12274.112} C_VEL
LIN {X 0,Y 375.955,Z 165.654,A -85,B 0,C 180,E1 -12276.742,E2 -12276.742} C_VEL
LIN {X 0,Y 375.99,Z 165.651,A -85,B 0,C 180,E1 -12279.971,E2 -12279.971} C_VEL
LIN {X 0,Y 375.932,Z 165.653,A -85,B 0,C 180,E1 -12283.766,E2 -12283.766} C_VEL
LIN {X 0,Y 375.993,Z 165.778,A -85,B 0,C 180,E1 -12284.647,E2 -12284.647} C_VEL
LIN {X 0,Y 377.094,Z 171.712,A -85,B 0,C 180,E1 -12288.202,E2 -12288.202} C_VEL
LIN {X 0,Y 378.079,Z 177.231,A -85,B 0,C 180,E1 -12291.328,E2 -12291.328} C_VEL
LIN {X 0,Y 378.518,Z 181.388,A -85,B 0,C 180,E1 -12293.548,E2 -12293.548} C_VEL
LIN {X 0,Y 378.101,Z 186.504,A -85,B 0,C 180,E1 -12296.108,E2 -12296.108} C_VEL
LIN {X 0,Y 377.53,Z 192.289,A -85,B 0,C 180,E1 -12298.907,E2 -12298.907} C_VEL
LIN {X 0,Y 376.762,Z 200.606,A -85,B 0,C 180,E1 -12302.805,E2 -12302.805} C_VEL
LIN {X 0,Y 376.125,Z 208.277,A -85,B 0,C 180,E1 -12306.289,E2 -12306.289} C_VEL
LIN {X 0,Y 375.62,Z 216.186,A -85,B 0,C 180,E1 -12309.8,E2 -12309.8} C_VEL
LIN {X 0,Y 375.509,Z 218.423,A -85,B 0,C 180,E1 -12310.775,E2 -12310.775} C_VEL
LIN {X 0,Y 377.795,Z 232.077,A -85,B 0,C 180,E1 -12311.347,E2 -12311.347} C_VEL
LIN {X 0,Y 379.392,Z 244.588,A -85,B 0,C 180,E1 -12312.068,E2 -12312.068} C_VEL
LIN {X 0,Y 380.302,Z 253.483,A -85,B 0,C 180,E1 -12312.699,E2 -12312.699} C_VEL
LIN {X 0,Y 379.218,Z 265.966,A -85,B 0,C 180,E1 -12313.721,E2 -12313.721} C_VEL
LIN {X 0,Y 378.188,Z 277.401,A -85,B 0,C 180,E1 -12314.92,E2 -12314.92} C_VEL
LIN {X 0,Y 377.309,Z 287.539,A -85,B 0,C 180,E1 -12316.262,E2 -12316.262} C_VEL
LIN {X 0,Y 376.373,Z 297.329,A -85,B 0,C 180,E1 -12317.874,E2 -12317.874} C_VEL
LIN {X 0,Y 375.664,Z 305.176,A -85,B 0,C 180,E1 -12319.49,E2 -12319.49} C_VEL
LIN {X 0,Y 375.237,Z 310.521,A -85,B 0,C 180,E1 -12320.84,E2 -12320.84} C_VEL
LIN {X 0,Y 374.865,Z 315.724,A -85,B 0,C 180,E1 -12322.459,E2 -12322.459} C_VEL
LIN {X 0,Y 374.7,Z 319.047,A -85,B 0,C 180,E1 -12323.77,E2 -12323.77} C_VEL
LIN {X 0,Y 374.586,Z 322.735,A -85,B 0,C 180,E1 -12325.696,E2 -12325.696} C_VEL
LIN {X 0,Y 374.521,Z 324.159,A -85,B 0,C 180,E1 -12326.773,E2 -12326.773} C_VEL
LIN {X 0,Y 374.604,Z 325.171,A -85,B 0,C 180,E1 -12327.85,E2 -12327.85} C_VEL
LIN {X 0,Y 374.603,Z 325.782,A -85,B 0,C 180,E1 -12328.925,E2 -12328.925} C_VEL
LIN {X 0,Y 374.596,Z 325.998,A -85,B 0,C 180,E1 -12330,E2 -12330} C_VEL
LIN {X 0,Y 374.603,Z 325.777,A -85,B 0,C 180,E1 -12331.075,E2 -12331.075} C_VEL
LIN {X 0,Y 374.592,Z 325.146,A -85,B 0,C 180,E1 -12332.151,E2 -12332.151} C_VEL
LIN {X 0,Y 374.587,Z 322.693,A -85,B 0,C 180,E1 -12334.304,E2 -12334.304} C_VEL
LIN {X 0,Y 374.7,Z 319.001,A -85,B 0,C 180,E1 -12336.23,E2 -12336.23} C_VEL
LIN {X 0,Y 374.945,Z 314.047,A -85,B 0,C 180,E1 -12338.082,E2 -12338.082} C_VEL
LIN {X 0,Y 375.394,Z 308.451,A -85,B 0,C 180,E1 -12339.701,E2 -12339.701} C_VEL
LIN {X 0,Y 375.967,Z 301.483,A -85,B 0,C 180,E1 -12341.32,E2 -12341.32} C_VEL
LIN {X 0,Y 376.847,Z 292.818,A -85,B 0,C 180,E1 -12342.932,E2 -12342.932} C_VEL
LIN {X 0,Y 377.728,Z 283.552,A -85,B 0,C 180,E1 -12344.33,E2 -12344.33} C_VEL
LIN {X 0,Y 378.628,Z 273.112,A -85,B 0,C 180,E1 -12345.614,E2 -12345.614} C_VEL
LIN {X 0,Y 379.685,Z 262.305,A -85,B 0,C 180,E1 -12346.673,E2 -12346.673} C_VEL
LIN {X 0,Y 380.456,Z 252.925,A -85,B 0,C 180,E1 -12347.419,E2 -12347.419} C_VEL
LIN {X 0,Y 379.214,Z 241.186,A -85,B 0,C 180,E1 -12348.254,E2 -12348.254} C_VEL
LIN {X 0,Y 377.398,Z 227.571,A -85,B 0,C 180,E1 -12349.009,E2 -12349.009} C_VEL
LIN {X 0,Y 375.503,Z 217.169,A -85,B 0,C 180,E1 -12349.474,E2 -12349.474} C_VEL
LIN {X 0,Y 375.965,Z 208.93,A -85,B 0,C 180,E1 -12353.114,E2 -12353.114} C_VEL
LIN {X 0,Y 376.551,Z 201.263,A -85,B 0,C 180,E1 -12356.612,E2 -12356.612} C_VEL
LIN {X 0,Y 377.263,Z 193.687,A -85,B 0,C 180,E1 -12360.198,E2 -12360.198} C_VEL
LIN {X 0,Y 377.917,Z 187.659,A -85,B 0,C 180,E1 -12363.19,E2 -12363.19} C_VEL
LIN {X 0,Y 378.512,Z 182.698,A -85,B 0,C 180,E1 -12365.794,E2 -12365.794} C_VEL
LIN {X 0,Y 378.41,Z 179.169,A -85,B 0,C 180,E1 -12367.799,E2 -12367.799} C_VEL
LIN {X 0,Y 377.62,Z 174.565,A -85,B 0,C 180,E1 -12370.647,E2 -12370.647} C_VEL
LIN {X 0,Y 376.753,Z 170.138,A -85,B 0,C 180,E1 -12373.647,E2 -12373.647} C_VEL
LIN {X 0,Y 375.981,Z 165.656,A -85,B 0,C 180,E1 -12377.134,E2 -12377.134} C_VEL
LIN {X 0,Y 375.967,Z 165.657,A -85,B 0,C 180,E1 -12380.537,E2 -12380.537} C_VEL
LIN {X 0,Y 375.968,Z 165.655,A -85,B 0,C 180,E1 -12383.495,E2 -12383.495} C_VEL
LIN {X 0,Y 375.964,Z 165.653,A -85,B 0,C 180,E1 -12385.888,E2 -12385.888} C_VEL
LIN {X 0,Y 375.969,Z 165.654,A -85,B 0,C 180,E1 -12389.687,E2 -12389.687} C_VEL
LIN {X 0,Y 376.024,Z 165.645,A -85,B 0,C 180,E1 -12393.348,E2 -12393.348} C_VEL
LIN {X 0,Y 376.001,Z 165.65,A -85,B 0,C 180,E1 -12396.888,E2 -12396.888} C_VEL
LIN {X 0,Y 376.001,Z 165.649,A -85,B 0,C 180,E1 -12400.339,E2 -12400.339} C_VEL
LIN {X 0,Y 376.03,Z 165.646,A -85,B 0,C 180,E1 -12403.718,E2 -12403.718} C_VEL
LIN {X 0,Y 376.108,Z 165.637,A -85,B 0,C 180,E1 -12407.042,E2 -12407.042} C_VEL
LIN {X 0,Y 376.124,Z 165.636,A -85,B 0,C 180,E1 -12410.318,E2 -12410.318} C_VEL
LIN {X 0,Y 376.235,Z 165.622,A -85,B 0,C 180,E1 -12412.486,E2 -12412.486} C_VEL
LIN {X 0,Y 376.176,Z 165.63,A -85,B 0,C 180,E1 -12414.639,E2 -12414.639} C_VEL
LIN {X 0,Y 376.358,Z 165.605,A -85,B 0,C 180,E1 -12417.859,E2 -12417.859} C_VEL
LIN {X 0,Y 376.493,Z 165.59,A -85,B 0,C 180,E1 -12419.999,E2 -12419.999} C_VEL
LIN {X 0,Y 376.192,Z 165.627,A -85,B 0,C 180,E1 -12423.212,E2 -12423.212} C_VEL
LIN {X 0,Y 376.225,Z 165.626,A -85,B 0,C 180,E1 -12426.583,E2 -12426.583} C_VEL
LIN {X 0,Y 376.094,Z 165.641,A -85,B 0,C 180,E1 -12428.597,E2 -12428.597} C_VEL
LIN {X 0,Y 376.004,Z 165.699,A -85,B 0,C 180,E1 -12429.684,E2 -12429.684} C_VEL
LIN {X 0,Y 375.906,Z 168.863,A -85,B 0,C 180,E1 -12433.54,E2 -12433.54} C_VEL
LIN {X 0,Y 375.654,Z 172.229,A -85,B 0,C 180,E1 -12437.417,E2 -12437.417} C_VEL
LIN {X 0,Y 375.44,Z 175.232,A -85,B 0,C 180,E1 -12440.834,E2 -12440.834} C_VEL
LIN {X 0,Y 375.343,Z 177.593,A -85,B 0,C 180,E1 -12443.438,E2 -12443.438} C_VEL
LIN {X 0,Y 375.32,Z 179.777,A -85,B 0,C 180,E1 -12445.623,E2 -12445.623} C_VEL
LIN {X 0,Y 379.441,Z 193.509,A -85,B 0,C 180,E1 -12446.441,E2 -12446.441} C_VEL
LIN {X 0,Y 381.931,Z 204.346,A -85,B 0,C 180,E1 -12447.216,E2 -12447.216} C_VEL
LIN {X 0,Y 381.198,Z 215.884,A -85,B 0,C 180,E1 -12448.048,E2 -12448.048} C_VEL
LIN {X 0,Y 380.184,Z 227.604,A -85,B 0,C 180,E1 -12449.139,E2 -12449.139} C_VEL
LIN {X 0,Y 379.324,Z 237.702,A -85,B 0,C 180,E1 -12450.323,E2 -12450.323} C_VEL
LIN {X 0,Y 378.384,Z 246.922,A -85,B 0,C 180,E1 -12451.647,E2 -12451.647} C_VEL
LIN {X 0,Y 377.405,Z 255.859,A -85,B 0,C 180,E1 -12453.251,E2 -12453.251} C_VEL
LIN {X 0,Y 376.467,Z 263.787,A -85,B 0,C 180,E1 -12455.037,E2 -12455.037} C_VEL
LIN {X 0,Y 375.912,Z 269.649,A -85,B 0,C 180,E1 -12456.745,E2 -12456.745} C_VEL
LIN {X 0,Y 375.47,Z 273.549,A -85,B 0,C 180,E1 -12458.172,E2 -12458.172} C_VEL
LIN {X 0,Y 375.084,Z 276.948,A -85,B 0,C 180,E1 -12459.805,E2 -12459.805} C_VEL
LIN {X 0,Y 374.824,Z 279.285,A -85,B 0,C 180,E1 -12461.409,E2 -12461.409} C_VEL
LIN {X 0,Y 374.61,Z 280.663,A -85,B 0,C 180,E1 -12462.973,E2 -12462.973} C_VEL
LIN {X 0,Y 374.531,Z 281.186,A -85,B 0,C 180,E1 -12464.515,E2 -12464.515} C_VEL
LIN {X 0,Y 374.518,Z 280.913,A -85,B 0,C 180,E1 -12466.026,E2 -12466.026} C_VEL
LIN {X 0,Y 374.62,Z 279.88,A -85,B 0,C 180,E1 -12467.516,E2 -12467.516} C_VEL
LIN {X 0,Y 374.931,Z 276.993,A -85,B 0,C 180,E1 -12469.638,E2 -12469.638} C_VEL
LIN {X 0,Y 375.158,Z 273.972,A -85,B 0,C 180,E1 -12471.129,E2 -12471.129} C_VEL
LIN {X 0,Y 375.682,Z 268.168,A -85,B 0,C 180,E1 -12473.228,E2 -12473.228} C_VEL
LIN {X 0,Y 376.213,Z 261.731,A -85,B 0,C 180,E1 -12474.968,E2 -12474.968} C_VEL
LIN {X 0,Y 376.882,Z 254.573,A -85,B 0,C 180,E1 -12476.516,E2 -12476.516} C_VEL
LIN {X 0,Y 377.768,Z 246.231,A -85,B 0,C 180,E1 -12477.98,E2 -12477.98} C_VEL
LIN {X 0,Y 378.508,Z 237.091,A -85,B 0,C 180,E1 -12479.295,E2 -12479.295} C_VEL
LIN {X 0,Y 379.343,Z 226.3,A -85,B 0,C 180,E1 -12480.545,E2 -12480.545} C_VEL
LIN {X 0,Y 380.185,Z 214.843,A -85,B 0,C 180,E1 -12481.605,E2 -12481.605} C_VEL
LIN {X 0,Y 380.995,Z 203.17,A -85,B 0,C 180,E1 -12482.441,E2 -12482.441} C_VEL
LIN {X 0,Y 378.611,Z 191.544,A -85,B 0,C 180,E1 -12483.21,E2 -12483.21} C_VEL
LIN {X 0,Y 375.055,Z 177.399,A -85,B 0,C 180,E1 -12483.949,E2 -12483.949} C_VEL
LIN {X 0,Y 375.073,Z 174.466,A -85,B 0,C 180,E1 -12486.828,E2 -12486.828} C_VEL
LIN {X 0,Y 375.177,Z 170.995,A -85,B 0,C 180,E1 -12490.294,E2 -12490.294} C_VEL
LIN {X 0,Y 375.302,Z 167.655,A -85,B 0,C 180,E1 -12493.686,E2 -12493.686} C_VEL
LIN {X 0,Y 375.421,Z 165.724,A -85,B 0,C 180,E1 -12495.915,E2 -12495.915} C_VEL
LIN {X 0,Y 375.863,Z 165.664,A -85,B 0,C 180,E1 -12499.223,E2 -12499.223} C_VEL
LIN {X 0,Y 376.18,Z 165.628,A -85,B 0,C 180,E1 -12502.485,E2 -12502.485} C_VEL
LIN {X 0,Y 376.163,Z 165.628,A -85,B 0,C 180,E1 -12504.64,E2 -12504.64} C_VEL
LIN {X 0,Y 376.351,Z 165.607,A -85,B 0,C 180,E1 -12507.859,E2 -12507.859} C_VEL
LIN {X 0,Y 376.486,Z 165.591,A -85,B 0,C 180,E1 -12510,E2 -12510} C_VEL
LIN {X 0,Y 376.186,Z 165.624,A -85,B 0,C 180,E1 -12513.213,E2 -12513.213} C_VEL
LIN {X 0,Y 376.242,Z 165.618,A -85,B 0,C 180,E1 -12516.435,E2 -12516.435} C_VEL
LIN {X 0,Y 376.202,Z 165.622,A -85,B 0,C 180,E1 -12518.595,E2 -12518.595} C_VEL
LIN {X 0,Y 376.047,Z 165.646,A -85,B 0,C 180,E1 -12521.863,E2 -12521.863} C_VEL
LIN {X 0,Y 376.055,Z 165.642,A -85,B 0,C 180,E1 -12525.167,E2 -12525.167} C_VEL
LIN {X 0,Y 376.005,Z 165.646,A -85,B 0,C 180,E1 -12528.527,E2 -12528.527} C_VEL
LIN {X 0,Y 375.96,Z 165.654,A -85,B 0,C 180,E1 -12531.954,E2 -12531.954} C_VEL
LIN {X 0,Y 376.003,Z 165.651,A -85,B 0,C 180,E1 -12535.461,E2 -12535.461} C_VEL
LIN {X 0,Y 376.016,Z 165.646,A -85,B 0,C 180,E1 -12535.908,E2 -12535.908} C_VEL
LIN {X 0,Y 375.372,Z 165.728,A -85,B 0,C 180,E1 -12536.802,E2 -12536.802} C_VEL
LIN {X 0,Y 372.472,Z 166.086,A -85,B 0,C 180,E1 -12538.255,E2 -12538.255} C_VEL
LIN {X 0,Y 370.01,Z 166.397,A -85,B 0,C 180,E1 -12539.43,E2 -12539.43} C_VEL
LIN {X 0,Y 368.976,Z 166.522,A -85,B 0,C 180,E1 -12540.34,E2 -12540.34} C_VEL
LIN {X 0,Y 368.906,Z 166.531,A -85,B 0,C 180,E1 -12540.648,E2 -12540.648} C_VEL
LIN {X 0,Y 368.893,Z 166.535,A -85,B 0,C 180,E1 -12543.538,E2 -12543.538} C_VEL
LIN {X 0,Y 368.898,Z 166.534,A -85,B 0,C 180,E1 -12546.856,E2 -12546.856} C_VEL
LIN {X 0,Y 368.908,Z 166.53,A -85,B 0,C 180,E1 -12550.37,E2 -12550.37} C_VEL
LIN {X 0,Y 368.881,Z 166.534,A -85,B 0,C 180,E1 -12553.617,E2 -12553.617} C_VEL
LIN {X 0,Y 368.883,Z 166.537,A -85,B 0,C 180,E1 -12556.696,E2 -12556.696} C_VEL
LIN {X 0,Y 368.909,Z 166.53,A -85,B 0,C 180,E1 -12559.643,E2 -12559.643} C_VEL
LIN {X 0,Y 368.901,Z 166.534,A -85,B 0,C 180,E1 -12563.144,E2 -12563.144} C_VEL
LIN {X 0,Y 368.894,Z 166.535,A -85,B 0,C 180,E1 -12566.462,E2 -12566.462} C_VEL
LIN {X 0,Y 368.927,Z 166.53,A -85,B 0,C 180,E1 -12569.047,E2 -12569.047} C_VEL
LIN {X 0,Y 368.962,Z 166.528,A -85,B 0,C 180,E1 -12572.797,E2 -12572.797} C_VEL
LIN {X 0,Y 368.945,Z 166.527,A -85,B 0,C 180,E1 -12576.113,E2 -12576.113} C_VEL
LIN {X 0,Y 368.936,Z 166.528,A -85,B 0,C 180,E1 -12579.948,E2 -12579.948} C_VEL
LIN {X 0,Y 368.975,Z 166.522,A -85,B 0,C 180,E1 -12583.399,E2 -12583.399} C_VEL
LIN {X 0,Y 369.058,Z 166.514,A -85,B 0,C 180,E1 -12586.791,E2 -12586.791} C_VEL
LIN {X 0,Y 369.068,Z 166.515,A -85,B 0,C 180,E1 -12590.132,E2 -12590.132} C_VEL
LIN {X 0,Y 369.197,Z 166.495,A -85,B 0,C 180,E1 -12593.442,E2 -12593.442} C_VEL
LIN {X 0,Y 369.32,Z 166.482,A -85,B 0,C 180,E1 -12597.819,E2 -12597.819} C_VEL
LIN {X 0,Y 369.458,Z 166.466,A -85,B 0,C 180,E1 -12600.001,E2 -12600.001} C_VEL
LIN {X 0,Y 369.318,Z 166.483,A -85,B 0,C 180,E1 -12602.182,E2 -12602.182} C_VEL
LIN {X 0,Y 369.175,Z 166.498,A -85,B 0,C 180,E1 -12606.559,E2 -12606.559} C_VEL
LIN {X 0,Y 369.065,Z 166.515,A -85,B 0,C 180,E1 -12609.869,E2 -12609.869} C_VEL
LIN {X 0,Y 369.039,Z 166.519,A -85,B 0,C 180,E1 -12613.773,E2 -12613.773} C_VEL
LIN {X 0,Y 369.003,Z 166.523,A -85,B 0,C 180,E1 -12617.769,E2 -12617.769} C_VEL
LIN {X 0,Y 368.931,Z 166.53,A -85,B 0,C 180,E1 -12621.22,E2 -12621.22} C_VEL
LIN {X 0,Y 368.96,Z 166.524,A -85,B 0,C 180,E1 -12624.776,E2 -12624.776} C_VEL
LIN {X 0,Y 368.965,Z 166.526,A -85,B 0,C 180,E1 -12627.204,E2 -12627.204} C_VEL
LIN {X 0,Y 368.931,Z 166.529,A -85,B 0,C 180,E1 -12630.954,E2 -12630.954} C_VEL
LIN {X 0,Y 368.931,Z 166.531,A -85,B 0,C 180,E1 -12635.002,E2 -12635.002} C_VEL
LIN {X 0,Y 368.91,Z 166.532,A -85,B 0,C 180,E1 -12638.64,E2 -12638.64} C_VEL
LIN {X 0,Y 368.883,Z 166.533,A -85,B 0,C 180,E1 -12642.01,E2 -12642.01} C_VEL
LIN {X 0,Y 368.956,Z 166.737,A -85,B 0,C 180,E1 -12644.324,E2 -12644.324} C_VEL
LIN {X 0,Y 370.009,Z 172.383,A -85,B 0,C 180,E1 -12647.798,E2 -12647.798} C_VEL
LIN {X 0,Y 371.104,Z 178.487,A -85,B 0,C 180,E1 -12651.321,E2 -12651.321} C_VEL
LIN {X 0,Y 371.511,Z 182.362,A -85,B 0,C 180,E1 -12653.424,E2 -12653.424} C_VEL
LIN {X 0,Y 370.997,Z 188.305,A -85,B 0,C 180,E1 -12656.462,E2 -12656.462} C_VEL
LIN {X 0,Y 370.4,Z 193.853,A -85,B 0,C 180,E1 -12659.183,E2 -12659.183} C_VEL
LIN {X 0,Y 369.816,Z 200.243,A -85,B 0,C 180,E1 -12662.251,E2 -12662.251} C_VEL
LIN {X 0,Y 369.077,Z 208.458,A -85,B 0,C 180,E1 -12666.068,E2 -12666.068} C_VEL
LIN {X 0,Y 368.638,Z 215.091,A -85,B 0,C 180,E1 -12669.096,E2 -12669.096} C_VEL
LIN {X 0,Y 368.46,Z 217.975,A -85,B 0,C 180,E1 -12670.393,E2 -12670.393} C_VEL
LIN {X 0,Y 371.037,Z 233.484,A -85,B 0,C 180,E1 -12671.105,E2 -12671.105} C_VEL
LIN {X 0,Y 372.75,Z 247.261,A -85,B 0,C 180,E1 -12671.954,E2 -12671.954} C_VEL
LIN {X 0,Y 373.383,Z 254.132,A -85,B 0,C 180,E1 -12672.473,E2 -12672.473} C_VEL
LIN {X 0,Y 372.357,Z 265.34,A -85,B 0,C 180,E1 -12673.413,E2 -12673.413} C_VEL
LIN {X 0,Y 371.286,Z 276.81,A -85,B 0,C 180,E1 -12674.633,E2 -12674.633} C_VEL
LIN {X 0,Y 370.586,Z 285.124,A -85,B 0,C 180,E1 -12675.727,E2 -12675.727} C_VEL
LIN {X 0,Y 369.723,Z 293.796,A -85,B 0,C 180,E1 -12677.094,E2 -12677.094} C_VEL
LIN {X 0,Y 368.834,Z 302.22,A -85,B 0,C 180,E1 -12678.737,E2 -12678.737} C_VEL
LIN {X 0,Y 368.256,Z 309.012,A -85,B 0,C 180,E1 -12680.387,E2 -12680.387} C_VEL
LIN {X 0,Y 367.783,Z 315.25,A -85,B 0,C 180,E1 -12682.313,E2 -12682.313} C_VEL
LIN {X 0,Y 367.601,Z 318.954,A -85,B 0,C 180,E1 -12683.811,E2 -12683.811} C_VEL
LIN {X 0,Y 367.517,Z 322.288,A -85,B 0,C 180,E1 -12685.613,E2 -12685.613} C_VEL
LIN {X 0,Y 367.435,Z 323.723,A -85,B 0,C 180,E1 -12686.711,E2 -12686.711} C_VEL
LIN {X 0,Y 367.507,Z 324.739,A -85,B 0,C 180,E1 -12687.808,E2 -12687.808} C_VEL
LIN {X 0,Y 367.539,Z 325.356,A -85,B 0,C 180,E1 -12688.905,E2 -12688.905} C_VEL
LIN {X 0,Y 367.53,Z 325.576,A -85,B 0,C 180,E1 -12690,E2 -12690} C_VEL
LIN {X 0,Y 367.538,Z 325.364,A -85,B 0,C 180,E1 -12691.096,E2 -12691.096} C_VEL
LIN {X 0,Y 367.495,Z 324.735,A -85,B 0,C 180,E1 -12692.192,E2 -12692.192} C_VEL
LIN {X 0,Y 367.517,Z 322.289,A -85,B 0,C 180,E1 -12694.387,E2 -12694.387} C_VEL
LIN {X 0,Y 367.597,Z 318.995,A -85,B 0,C 180,E1 -12696.182,E2 -12696.182} C_VEL
LIN {X 0,Y 367.894,Z 313.662,A -85,B 0,C 180,E1 -12698.238,E2 -12698.238} C_VEL
LIN {X 0,Y 368.428,Z 307.049,A -85,B 0,C 180,E1 -12700.163,E2 -12700.163} C_VEL
LIN {X 0,Y 369.085,Z 299.816,A -85,B 0,C 180,E1 -12701.812,E2 -12701.812} C_VEL
LIN {X 0,Y 370.076,Z 290.856,A -85,B 0,C 180,E1 -12703.453,E2 -12703.453} C_VEL
LIN {X 0,Y 370.917,Z 281.686,A -85,B 0,C 180,E1 -12704.823,E2 -12704.823} C_VEL
LIN {X 0,Y 371.9,Z 271.653,A -85,B 0,C 180,E1 -12706.044,E2 -12706.044} C_VEL
LIN {X 0,Y 373.021,Z 260.572,A -85,B 0,C 180,E1 -12707.121,E2 -12707.121} C_VEL
LIN {X 0,Y 373.592,Z 252.888,A -85,B 0,C 180,E1 -12707.744,E2 -12707.744} C_VEL
LIN {X 0,Y 372.377,Z 241.486,A -85,B 0,C 180,E1 -12708.59,E2 -12708.59} C_VEL
LIN {X 0,Y 370.55,Z 227.733,A -85,B 0,C 180,E1 -12709.385,E2 -12709.385} C_VEL
LIN {X 0,Y 368.474,Z 216.711,A -85,B 0,C 180,E1 -12709.898,E2 -12709.898} C_VEL
LIN {X 0,Y 369.017,Z 207.881,A -85,B 0,C 180,E1 -12713.911,E2 -12713.911} C_VEL
LIN {X 0,Y 369.735,Z 199.728,A -85,B 0,C 180,E1 -12717.756,E2 -12717.756} C_VEL
LIN {X 0,Y 370.481,Z 192.367,A -85,B 0,C 180,E1 -12721.389,E2 -12721.389} C_VEL
LIN {X 0,Y 371.24,Z 186.174,A -85,B 0,C 180,E1 -12724.607,E2 -12724.607} C_VEL
LIN {X 0,Y 371.564,Z 182.597,A -85,B 0,C 180,E1 -12726.571,E2 -12726.571} C_VEL
LIN {X 0,Y 371.075,Z 178.463,A -85,B 0,C 180,E1 -12729.056,E2 -12729.056} C_VEL
LIN {X 0,Y 370.234,Z 173.653,A -85,B 0,C 180,E1 -12732.241,E2 -12732.241} C_VEL
LIN {X 0,Y 369.452,Z 169.502,A -85,B 0,C 180,E1 -12735.263,E2 -12735.263} C_VEL
LIN {X 0,Y 368.913,Z 166.538,A -85,B 0,C 180,E1 -12737.74,E2 -12737.74} C_VEL
LIN {X 0,Y 368.913,Z 166.536,A -85,B 0,C 180,E1 -12741.359,E2 -12741.359} C_VEL
LIN {X 0,Y 368.941,Z 166.53,A -85,B 0,C 180,E1 -12745.146,E2 -12745.146} C_VEL
LIN {X 0,Y 368.933,Z 166.529,A -85,B 0,C 180,E1 -12749.046,E2 -12749.046} C_VEL
LIN {X 0,Y 368.973,Z 166.524,A -85,B 0,C 180,E1 -12752.797,E2 -12752.797} C_VEL
LIN {X 0,Y 368.971,Z 166.527,A -85,B 0,C 180,E1 -12756.421,E2 -12756.421} C_VEL
LIN {X 0,Y 368.94,Z 166.527,A -85,B 0,C 180,E1 -12759.947,E2 -12759.947} C_VEL
LIN {X 0,Y 368.973,Z 166.526,A -85,B 0,C 180,E1 -12763.398,E2 -12763.398} C_VEL
LIN {X 0,Y 369.062,Z 166.515,A -85,B 0,C 180,E1 -12766.79,E2 -12766.79} C_VEL
LIN {X 0,Y 369.072,Z 166.514,A -85,B 0,C 180,E1 -12770.131,E2 -12770.131} C_VEL
LIN {X 0,Y 369.193,Z 166.499,A -85,B 0,C 180,E1 -12772.342,E2 -12772.342} C_VEL
LIN {X 0,Y 369.149,Z 166.505,A -85,B 0,C 180,E1 -12774.537,E2 -12774.537} C_VEL
LIN {X 0,Y 369.323,Z 166.481,A -85,B 0,C 180,E1 -12777.818,E2 -12777.818} C_VEL
LIN {X 0,Y 369.463,Z 166.466,A -85,B 0,C 180,E1 -12779.999,E2 -12779.999} C_VEL
LIN {X 0,Y 369.322,Z 166.482,A -85,B 0,C 180,E1 -12782.181,E2 -12782.181} C_VEL
LIN {X 0,Y 369.197,Z 166.502,A -85,B 0,C 180,E1 -12786.565,E2 -12786.565} C_VEL
LIN {X 0,Y 369.026,Z 166.521,A -85,B 0,C 180,E1 -12788.763,E2 -12788.763} C_VEL
LIN {X 0,Y 369.006,Z 166.967,A -85,B 0,C 180,E1 -12789.869,E2 -12789.869} C_VEL
LIN {X 0,Y 368.87,Z 170.038,A -85,B 0,C 180,E1 -12793.664,E2 -12793.664} C_VEL
LIN {X 0,Y 368.601,Z 173.357,A -85,B 0,C 180,E1 -12797.572,E2 -12797.572} C_VEL
LIN {X 0,Y 368.382,Z 176.553,A -85,B 0,C 180,E1 -12801.252,E2 -12801.252} C_VEL
LIN {X 0,Y 368.246,Z 180.028,A -85,B 0,C 180,E1 -12805.127,E2 -12805.127} C_VEL
LIN {X 0,Y 368.422,Z 181.03,A -85,B 0,C 180,E1 -12805.228,E2 -12805.228} C_VEL
LIN {X 0,Y 372.49,Z 193.937,A -85,B 0,C 180,E1 -12806.037,E2 -12806.037} C_VEL
LIN {X 0,Y 375.108,Z 205.14,A -85,B 0,C 180,E1 -12806.869,E2 -12806.869} C_VEL
LIN {X 0,Y 374.451,Z 216.698,A -85,B 0,C 180,E1 -12807.735,E2 -12807.735} C_VEL
LIN {X 0,Y 373.422,Z 228.226,A -85,B 0,C 180,E1 -12808.833,E2 -12808.833} C_VEL
LIN {X 0,Y 372.415,Z 239.141,A -85,B 0,C 180,E1 -12810.146,E2 -12810.146} C_VEL
LIN {X 0,Y 371.358,Z 248.821,A -85,B 0,C 180,E1 -12811.61,E2 -12811.61} C_VEL
LIN {X 0,Y 370.485,Z 256.458,A -85,B 0,C 180,E1 -12813.028,E2 -12813.028} C_VEL
LIN {X 0,Y 369.507,Z 264.143,A -85,B 0,C 180,E1 -12814.791,E2 -12814.791} C_VEL
LIN {X 0,Y 369.048,Z 268.943,A -85,B 0,C 180,E1 -12816.181,E2 -12816.181} C_VEL
LIN {X 0,Y 368.429,Z 274.102,A -85,B 0,C 180,E1 -12818.06,E2 -12818.06} C_VEL
LIN {X 0,Y 367.93,Z 278.179,A -85,B 0,C 180,E1 -12820.176,E2 -12820.176} C_VEL
LIN {X 0,Y 367.653,Z 280.406,A -85,B 0,C 180,E1 -12821.993,E2 -12821.993} C_VEL
LIN {X 0,Y 367.482,Z 281.392,A -85,B 0,C 180,E1 -12823.51,E2 -12823.51} C_VEL
LIN {X 0,Y 367.435,Z 281.619,A -85,B 0,C 180,E1 -12825.048,E2 -12825.048} C_VEL
LIN {X 0,Y 367.454,Z 281.042,A -85,B 0,C 180,E1 -12826.618,E2 -12826.618} C_VEL
LIN {X 0,Y 367.624,Z 279.582,A -85,B 0,C 180,E1 -12828.208,E2 -12828.208} C_VEL
LIN {X 0,Y 367.888,Z 277.191,A -85,B 0,C 180,E1 -12829.83,E2 -12829.83} C_VEL
LIN {X 0,Y 368.148,Z 273.717,A -85,B 0,C 180,E1 -12831.507,E2 -12831.507} C_VEL
LIN {X 0,Y 368.602,Z 269.042,A -85,B 0,C 180,E1 -12833.205,E2 -12833.205} C_VEL
LIN {X 0,Y 369.138,Z 262.864,A -85,B 0,C 180,E1 -12834.951,E2 -12834.951} C_VEL
LIN {X 0,Y 369.917,Z 254.921,A -85,B 0,C 180,E1 -12836.714,E2 -12836.714} C_VEL
LIN {X 0,Y 370.87,Z 246.225,A -85,B 0,C 180,E1 -12838.26,E2 -12838.26} C_VEL
LIN {X 0,Y 371.721,Z 236.113,A -85,B 0,C 180,E1 -12839.707,E2 -12839.707} C_VEL
LIN {X 0,Y 372.594,Z 225.391,A -85,B 0,C 180,E1 -12840.941,E2 -12840.941} C_VEL
LIN {X 0,Y 373.418,Z 214.646,A -85,B 0,C 180,E1 -12841.932,E2 -12841.932} C_VEL
LIN {X 0,Y 374.078,Z 203.457,A -85,B 0,C 180,E1 -12842.745,E2 -12842.745} C_VEL
LIN {X 0,Y 371.176,Z 190.103,A -85,B 0,C 180,E1 -12843.64,E2 -12843.64} C_VEL
LIN {X 0,Y 368.024,Z 177.786,A -85,B 0,C 180,E1 -12844.288,E2 -12844.288} C_VEL
LIN {X 0,Y 368.007,Z 174.509,A -85,B 0,C 180,E1 -12847.545,E2 -12847.545} C_VEL
LIN {X 0,Y 368.115,Z 171.05,A -85,B 0,C 180,E1 -12851.061,E2 -12851.061} C_VEL
LIN {X 0,Y 368.278,Z 167.698,A -85,B 0,C 180,E1 -12854.504,E2 -12854.504} C_VEL
LIN {X 0,Y 368.335,Z 166.634,A -85,B 0,C 180,E1 -12855.638,E2 -12855.638} C_VEL
LIN {X 0,Y 368.791,Z 166.545,A -85,B 0,C 180,E1 -12859.014,E2 -12859.014} C_VEL
LIN {X 0,Y 369.132,Z 166.507,A -85,B 0,C 180,E1 -12862.341,E2 -12862.341} C_VEL
LIN {X 0,Y 369.135,Z 166.504,A -85,B 0,C 180,E1 -12864.537,E2 -12864.537} C_VEL
LIN {X 0,Y 369.316,Z 166.483,A -85,B 0,C 180,E1 -12867.819,E2 -12867.819} C_VEL
LIN {X 0,Y 369.455,Z 166.467,A -85,B 0,C 180,E1 -12870,E2 -12870} C_VEL
LIN {X 0,Y 369.316,Z 166.483,A -85,B 0,C 180,E1 -12872.181,E2 -12872.181} C_VEL
LIN {X 0,Y 369.203,Z 166.494,A -85,B 0,C 180,E1 -12876.558,E2 -12876.558} C_VEL
LIN {X 0,Y 369.134,Z 166.502,A -85,B 0,C 180,E1 -12878.761,E2 -12878.761} C_VEL
LIN {X 0,Y 369.002,Z 166.521,A -85,B 0,C 180,E1 -12882.093,E2 -12882.093} C_VEL
LIN {X 0,Y 368.994,Z 166.523,A -85,B 0,C 180,E1 -12885.465,E2 -12885.465} C_VEL
LIN {X 0,Y 368.955,Z 166.524,A -85,B 0,C 180,E1 -12888.894,E2 -12888.894} C_VEL
LIN {X 0,Y 368.929,Z 166.528,A -85,B 0,C 180,E1 -12892.395,E2 -12892.395} C_VEL
LIN {X 0,Y 368.997,Z 166.521,A -85,B 0,C 180,E1 -12895.98,E2 -12895.98} C_VEL
LIN {X 0,Y 368.911,Z 166.533,A -85,B 0,C 180,E1 -12899.691,E2 -12899.691} C_VEL
LIN {X 0,Y 368.906,Z 166.531,A -85,B 0,C 180,E1 -12900.648,E2 -12900.648} C_VEL
LIN {X 0,Y 368.277,Z 166.614,A -85,B 0,C 180,E1 -12901.559,E2 -12901.559} C_VEL
LIN {X 0,Y 365.438,Z 166.972,A -85,B 0,C 180,E1 -12903.04,E2 -12903.04} C_VEL
LIN {X 0,Y 363.007,Z 167.275,A -85,B 0,C 180,E1 -12904.239,E2 -12904.239} C_VEL
LIN {X 0,Y 361.955,Z 167.402,A -85,B 0,C 180,E1 -12905.166,E2 -12905.166} C_VEL
LIN {X 0,Y 361.867,Z 167.41,A -85,B 0,C 180,E1 -12905.48,E2 -12905.48} C_VEL
LIN {X 0,Y 361.867,Z 167.412,A -85,B 0,C 180,E1 -12909.027,E2 -12909.027} C_VEL
LIN {X 0,Y 361.834,Z 167.415,A -85,B 0,C 180,E1 -12912.829,E2 -12912.829} C_VEL
LIN {X 0,Y 361.825,Z 167.412,A -85,B 0,C 180,E1 -12915.945,E2 -12915.945} C_VEL
LIN {X 0,Y 361.834,Z 167.414,A -85,B 0,C 180,E1 -12919.245,E2 -12919.245} C_VEL
LIN {X 0,Y 361.863,Z 167.412,A -85,B 0,C 180,E1 -12922.777,E2 -12922.777} C_VEL
LIN {X 0,Y 361.852,Z 167.409,A -85,B 0,C 180,E1 -12925.72,E2 -12925.72} C_VEL
LIN {X 0,Y 361.871,Z 167.406,A -85,B 0,C 180,E1 -12929.673,E2 -12929.673} C_VEL
LIN {X 0,Y 361.953,Z 167.396,A -85,B 0,C 180,E1 -12933.476,E2 -12933.476} C_VEL
LIN {X 0,Y 361.891,Z 167.405,A -85,B 0,C 180,E1 -12937.145,E2 -12937.145} C_VEL
LIN {X 0,Y 361.906,Z 167.406,A -85,B 0,C 180,E1 -12940.724,E2 -12940.724} C_VEL
LIN {X 0,Y 361.932,Z 167.4,A -85,B 0,C 180,E1 -12943.067,E2 -12943.067} C_VEL
LIN {X 0,Y 361.999,Z 167.395,A -85,B 0,C 180,E1 -12946.528,E2 -12946.528} C_VEL
LIN {X 0,Y 362.032,Z 167.389,A -85,B 0,C 180,E1 -12949.939,E2 -12949.939} C_VEL
LIN {X 0,Y 362.159,Z 167.371,A -85,B 0,C 180,E1 -12953.314,E2 -12953.314} C_VEL
LIN {X 0,Y 362.284,Z 167.358,A -85,B 0,C 180,E1 -12957.777,E2 -12957.777} C_VEL
LIN {X 0,Y 362.428,Z 167.342,A -85,B 0,C 180,E1 -12960.001,E2 -12960.001} C_VEL
LIN {X 0,Y 362.282,Z 167.359,A -85,B 0,C 180,E1 -12962.224,E2 -12962.224} C_VEL
LIN {X 0,Y 362.137,Z 167.374,A -85,B 0,C 180,E1 -12966.687,E2 -12966.687} C_VEL
LIN {X 0,Y 362.002,Z 167.394,A -85,B 0,C 180,E1 -12970.063,E2 -12970.063} C_VEL
LIN {X 0,Y 362,Z 167.395,A -85,B 0,C 180,E1 -12973.899,E2 -12973.899} C_VEL
LIN {X 0,Y 361.969,Z 167.398,A -85,B 0,C 180,E1 -12977.939,E2 -12977.939} C_VEL
LIN {X 0,Y 361.894,Z 167.408,A -85,B 0,C 180,E1 -12981.653,E2 -12981.653} C_VEL
LIN {X 0,Y 361.931,Z 167.403,A -85,B 0,C 180,E1 -12985.29,E2 -12985.29} C_VEL
LIN {X 0,Y 361.91,Z 167.404,A -85,B 0,C 180,E1 -12987.779,E2 -12987.779} C_VEL
LIN {X 0,Y 361.84,Z 167.414,A -85,B 0,C 180,E1 -12991.63,E2 -12991.63} C_VEL
LIN {X 0,Y 361.876,Z 167.411,A -85,B 0,C 180,E1 -12995.345,E2 -12995.345} C_VEL
LIN {X 0,Y 361.871,Z 167.411,A -85,B 0,C 180,E1 -12999.027,E2 -12999.027} C_VEL
LIN {X 0,Y 361.838,Z 167.41,A -85,B 0,C 180,E1 -13002.829,E2 -13002.829} C_VEL
LIN {X 0,Y 361.865,Z 167.481,A -85,B 0,C 180,E1 -13003.866,E2 -13003.866} C_VEL
LIN {X 0,Y 362.921,Z 173.066,A -85,B 0,C 180,E1 -13007.382,E2 -13007.382} C_VEL
LIN {X 0,Y 363.888,Z 178.451,A -85,B 0,C 180,E1 -13010.584,E2 -13010.584} C_VEL
LIN {X 0,Y 364.502,Z 183.276,A -85,B 0,C 180,E1 -13013.294,E2 -13013.294} C_VEL
LIN {X 0,Y 364.05,Z 188.673,A -85,B 0,C 180,E1 -13016.112,E2 -13016.112} C_VEL
LIN {X 0,Y 363.351,Z 194.758,A -85,B 0,C 180,E1 -13019.165,E2 -13019.165} C_VEL
LIN {X 0,Y 362.751,Z 201.14,A -85,B 0,C 180,E1 -13022.291,E2 -13022.291} C_VEL
LIN {X 0,Y 362.025,Z 208.811,A -85,B 0,C 180,E1 -13025.941,E2 -13025.941} C_VEL
LIN {X 0,Y 361.464,Z 217.142,A -85,B 0,C 180,E1 -13029.811,E2 -13029.811} C_VEL
LIN {X 0,Y 361.426,Z 217.672,A -85,B 0,C 180,E1 -13030.055,E2 -13030.055} C_VEL
LIN {X 0,Y 363.722,Z 231.231,A -85,B 0,C 180,E1 -13030.652,E2 -13030.652} C_VEL
LIN {X 0,Y 365.394,Z 243.948,A -85,B 0,C 180,E1 -13031.421,E2 -13031.421} C_VEL
LIN {X 0,Y 366.46,Z 255.139,A -85,B 0,C 180,E1 -13032.275,E2 -13032.275} C_VEL
LIN {X 0,Y 365.259,Z 267.49,A -85,B 0,C 180,E1 -13033.369,E2 -13033.369} C_VEL
LIN {X 0,Y 364.26,Z 277.717,A -85,B 0,C 180,E1 -13034.526,E2 -13034.526} C_VEL
LIN {X 0,Y 363.474,Z 286.413,A -85,B 0,C 180,E1 -13035.728,E2 -13035.728} C_VEL
LIN {X 0,Y 362.59,Z 294.759,A -85,B 0,C 180,E1 -13037.121,E2 -13037.121} C_VEL
LIN {X 0,Y 361.681,Z 302.933,A -85,B 0,C 180,E1 -13038.795,E2 -13038.795} C_VEL
LIN {X 0,Y 361.117,Z 309.525,A -85,B 0,C 180,E1 -13040.478,E2 -13040.478} C_VEL
LIN {X 0,Y 360.719,Z 314.769,A -85,B 0,C 180,E1 -13042.162,E2 -13042.162} C_VEL
LIN {X 0,Y 360.519,Z 318.803,A -85,B 0,C 180,E1 -13043.83,E2 -13043.83} C_VEL
LIN {X 0,Y 360.448,Z 321.837,A -85,B 0,C 180,E1 -13045.527,E2 -13045.527} C_VEL
LIN {X 0,Y 360.354,Z 323.284,A -85,B 0,C 180,E1 -13046.646,E2 -13046.646} C_VEL
LIN {X 0,Y 360.411,Z 324.305,A -85,B 0,C 180,E1 -13047.765,E2 -13047.765} C_VEL
LIN {X 0,Y 360.476,Z 324.928,A -85,B 0,C 180,E1 -13048.883,E2 -13048.883} C_VEL
LIN {X 0,Y 360.466,Z 325.153,A -85,B 0,C 180,E1 -13050,E2 -13050} C_VEL
LIN {X 0,Y 360.475,Z 324.952,A -85,B 0,C 180,E1 -13051.117,E2 -13051.117} C_VEL
LIN {X 0,Y 360.399,Z 324.325,A -85,B 0,C 180,E1 -13052.235,E2 -13052.235} C_VEL
LIN {X 0,Y 360.426,Z 321.888,A -85,B 0,C 180,E1 -13054.474,E2 -13054.474} C_VEL
LIN {X 0,Y 360.522,Z 318.87,A -85,B 0,C 180,E1 -13056.175,E2 -13056.175} C_VEL
LIN {X 0,Y 360.72,Z 314.89,A -85,B 0,C 180,E1 -13057.839,E2 -13057.839} C_VEL
LIN {X 0,Y 361.223,Z 308.748,A -85,B 0,C 180,E1 -13059.802,E2 -13059.802} C_VEL
LIN {X 0,Y 361.849,Z 302.045,A -85,B 0,C 180,E1 -13061.483,E2 -13061.483} C_VEL
LIN {X 0,Y 362.779,Z 293.761,A -85,B 0,C 180,E1 -13063.158,E2 -13063.158} C_VEL
LIN {X 0,Y 363.783,Z 284.245,A -85,B 0,C 180,E1 -13064.71,E2 -13064.71} C_VEL
LIN {X 0,Y 364.788,Z 273.821,A -85,B 0,C 180,E1 -13066.078,E2 -13066.078} C_VEL
LIN {X 0,Y 366.075,Z 262.004,A -85,B 0,C 180,E1 -13067.312,E2 -13067.312} C_VEL
LIN {X 0,Y 366.767,Z 254.263,A -85,B 0,C 180,E1 -13067.967,E2 -13067.967} C_VEL
LIN {X 0,Y 365.571,Z 241.869,A -85,B 0,C 180,E1 -13068.935,E2 -13068.935} C_VEL
LIN {X 0,Y 363.892,Z 228.902,A -85,B 0,C 180,E1 -13069.729,E2 -13069.729} C_VEL
LIN {X 0,Y 361.478,Z 216.239,A -85,B 0,C 180,E1 -13070.353,E2 -13070.353} C_VEL
LIN {X 0,Y 362.088,Z 207.021,A -85,B 0,C 180,E1 -13074.664,E2 -13074.664} C_VEL
LIN {X 0,Y 362.793,Z 199.478,A -85,B 0,C 180,E1 -13078.334,E2 -13078.334} C_VEL
LIN {X 0,Y 363.54,Z 192.789,A -85,B 0,C 180,E1 -13081.721,E2 -13081.721} C_VEL
LIN {X 0,Y 364.405,Z 186.021,A -85,B 0,C 180,E1 -13085.352,E2 -13085.352} C_VEL
LIN {X 0,Y 364.592,Z 183.686,A -85,B 0,C 180,E1 -13086.696,E2 -13086.696} C_VEL
LIN {X 0,Y 364.205,Z 180.292,A -85,B 0,C 180,E1 -13088.773,E2 -13088.773} C_VEL
LIN {X 0,Y 363.387,Z 175.686,A -85,B 0,C 180,E1 -13091.855,E2 -13091.855} C_VEL
LIN {X 0,Y 362.386,Z 170.352,A -85,B 0,C 180,E1 -13095.854,E2 -13095.854} C_VEL
LIN {X 0,Y 361.852,Z 167.416,A -85,B 0,C 180,E1 -13098.383,E2 -13098.383} C_VEL
LIN {X 0,Y 361.873,Z 167.414,A -85,B 0,C 180,E1 -13101.575,E2 -13101.575} C_VEL
LIN {X 0,Y 361.878,Z 167.411,A -85,B 0,C 180,E1 -13104.655,E2 -13104.655} C_VEL
LIN {X 0,Y 361.842,Z 167.415,A -85,B 0,C 180,E1 -13108.37,E2 -13108.37} C_VEL
LIN {X 0,Y 361.917,Z 167.406,A -85,B 0,C 180,E1 -13112.221,E2 -13112.221} C_VEL
LIN {X 0,Y 361.933,Z 167.402,A -85,B 0,C 180,E1 -13114.71,E2 -13114.71} C_VEL
LIN {X 0,Y 361.896,Z 167.407,A -85,B 0,C 180,E1 -13118.347,E2 -13118.347} C_VEL
LIN {X 0,Y 361.924,Z 167.399,A -85,B 0,C 180,E1 -13122.084,E2 -13122.084} C_VEL
LIN {X 0,Y 361.966,Z 167.399,A -85,B 0,C 180,E1 -13125.379,E2 -13125.379} C_VEL
LIN {X 0,Y 361.976,Z 167.398,A -85,B 0,C 180,E1 -13128.804,E2 -13128.804} C_VEL
LIN {X 0,Y 362.156,Z 167.375,A -85,B 0,C 180,E1 -13132.192,E2 -13132.192} C_VEL
LIN {X 0,Y 362.123,Z 167.379,A -85,B 0,C 180,E1 -13134.431,E2 -13134.431} C_VEL
LIN {X 0,Y 362.287,Z 167.357,A -85,B 0,C 180,E1 -13137.776,E2 -13137.776} C_VEL
LIN {X 0,Y 362.432,Z 167.342,A -85,B 0,C 180,E1 -13139.999,E2 -13139.999} C_VEL
LIN {X 0,Y 362.286,Z 167.358,A -85,B 0,C 180,E1 -13142.223,E2 -13142.223} C_VEL
LIN {X 0,Y 362.158,Z 167.379,A -85,B 0,C 180,E1 -13146.686,E2 -13146.686} C_VEL
LIN {X 0,Y 361.969,Z 167.4,A -85,B 0,C 180,E1 -13148.935,E2 -13148.935} C_VEL
LIN {X 0,Y 361.873,Z 170.018,A -85,B 0,C 180,E1 -13152.335,E2 -13152.335} C_VEL
LIN {X 0,Y 361.734,Z 171.901,A -85,B 0,C 180,E1 -13154.629,E2 -13154.629} C_VEL
LIN {X 0,Y 361.537,Z 174.817,A -85,B 0,C 180,E1 -13158.121,E2 -13158.121} C_VEL
LIN {X 0,Y 361.321,Z 177.887,A -85,B 0,C 180,E1 -13161.688,E2 -13161.688} C_VEL
LIN {X 0,Y 361.205,Z 180.58,A -85,B 0,C 180,E1 -13164.728,E2 -13164.728} C_VEL
LIN {X 0,Y 365.566,Z 194.609,A -85,B 0,C 180,E1 -13165.63,E2 -13165.63} C_VEL
LIN {X 0,Y 368.297,Z 205.756,A -85,B 0,C 180,E1 -13166.49,E2 -13166.49} C_VEL
LIN {X 0,Y 368.429,Z 208.623,A -85,B 0,C 180,E1 -13166.709,E2 -13166.709} C_VEL
LIN {X 0,Y 367.545,Z 219.753,A -85,B 0,C 180,E1 -13167.602,E2 -13167.602} C_VEL
LIN {X 0,Y 366.534,Z 230.088,A -85,B 0,C 180,E1 -13168.643,E2 -13168.643} C_VEL
LIN {X 0,Y 365.643,Z 239.549,A -85,B 0,C 180,E1 -13169.824,E2 -13169.824} C_VEL
LIN {X 0,Y 364.601,Z 248.569,A -85,B 0,C 180,E1 -13171.2,E2 -13171.2} C_VEL
LIN {X 0,Y 363.592,Z 256.91,A -85,B 0,C 180,E1 -13172.766,E2 -13172.766} C_VEL
LIN {X 0,Y 362.59,Z 264.328,A -85,B 0,C 180,E1 -13174.493,E2 -13174.493} C_VEL
LIN {X 0,Y 361.928,Z 270.422,A -85,B 0,C 180,E1 -13176.316,E2 -13176.316} C_VEL
LIN {X 0,Y 361.444,Z 274.326,A -85,B 0,C 180,E1 -13177.794,E2 -13177.794} C_VEL
LIN {X 0,Y 361.154,Z 276.632,A -85,B 0,C 180,E1 -13178.886,E2 -13178.886} C_VEL
LIN {X 0,Y 360.806,Z 279.367,A -85,B 0,C 180,E1 -13180.565,E2 -13180.565} C_VEL
LIN {X 0,Y 360.544,Z 281.12,A -85,B 0,C 180,E1 -13182.206,E2 -13182.206} C_VEL
LIN {X 0,Y 360.388,Z 281.968,A -85,B 0,C 180,E1 -13183.817,E2 -13183.817} C_VEL
LIN {X 0,Y 360.354,Z 281.977,A -85,B 0,C 180,E1 -13185.403,E2 -13185.403} C_VEL
LIN {X 0,Y 360.384,Z 281.216,A -85,B 0,C 180,E1 -13186.956,E2 -13186.956} C_VEL
LIN {X 0,Y 360.591,Z 279.7,A -85,B 0,C 180,E1 -13188.496,E2 -13188.496} C_VEL
LIN {X 0,Y 360.94,Z 276.262,A -85,B 0,C 180,E1 -13190.618,E2 -13190.618} C_VEL
LIN {X 0,Y 361.248,Z 272.631,A -85,B 0,C 180,E1 -13192.206,E2 -13192.206} C_VEL
LIN {X 0,Y 361.774,Z 267.269,A -85,B 0,C 180,E1 -13194.009,E2 -13194.009} C_VEL
LIN {X 0,Y 362.421,Z 260.549,A -85,B 0,C 180,E1 -13195.78,E2 -13195.78} C_VEL
LIN {X 0,Y 363.28,Z 252.435,A -85,B 0,C 180,E1 -13197.467,E2 -13197.467} C_VEL
LIN {X 0,Y 364.252,Z 242.752,A -85,B 0,C 180,E1 -13199.088,E2 -13199.088} C_VEL
LIN {X 0,Y 365.143,Z 232.347,A -85,B 0,C 180,E1 -13200.479,E2 -13200.479} C_VEL
LIN {X 0,Y 366.096,Z 221.174,A -85,B 0,C 180,E1 -13201.672,E2 -13201.672} C_VEL
LIN {X 0,Y 366.997,Z 209.719,A -85,B 0,C 180,E1 -13202.638,E2 -13202.638} C_VEL
LIN {X 0,Y 367.268,Z 204.822,A -85,B 0,C 180,E1 -13202.985,E2 -13202.985} C_VEL
LIN {X 0,Y 364.521,Z 192.131,A -85,B 0,C 180,E1 -13203.873,E2 -13203.873} C_VEL
LIN {X 0,Y 360.967,Z 178.17,A -85,B 0,C 180,E1 -13204.638,E2 -13204.638} C_VEL
LIN {X 0,Y 360.984,Z 174.553,A -85,B 0,C 180,E1 -13208.29,E2 -13208.29} C_VEL
LIN {X 0,Y 361.098,Z 171.087,A -85,B 0,C 180,E1 -13211.856,E2 -13211.856} C_VEL
LIN {X 0,Y 361.269,Z 167.756,A -85,B 0,C 180,E1 -13215.351,E2 -13215.351} C_VEL
LIN {X 0,Y 361.578,Z 167.445,A -85,B 0,C 180,E1 -13217.654,E2 -13217.654} C_VEL
LIN {X 0,Y 361.951,Z 167.397,A -85,B 0,C 180,E1 -13221.063,E2 -13221.063} C_VEL
LIN {X 0,Y 362.144,Z 167.372,A -85,B 0,C 180,E1 -13223.313,E2 -13223.313} C_VEL
LIN {X 0,Y 362.28,Z 167.359,A -85,B 0,C 180,E1 -13227.776,E2 -13227.776} C_VEL
LIN {X 0,Y 362.425,Z 167.343,A -85,B 0,C 180,E1 -13230,E2 -13230} C_VEL
LIN {X 0,Y 362.28,Z 167.359,A -85,B 0,C 180,E1 -13232.223,E2 -13232.223} C_VEL
LIN {X 0,Y 362.167,Z 167.37,A -85,B 0,C 180,E1 -13236.686,E2 -13236.686} C_VEL
LIN {X 0,Y 362.071,Z 167.382,A -85,B 0,C 180,E1 -13238.933,E2 -13238.933} C_VEL
LIN {X 0,Y 361.957,Z 167.397,A -85,B 0,C 180,E1 -13242.332,E2 -13242.332} C_VEL
LIN {X 0,Y 361.958,Z 167.396,A -85,B 0,C 180,E1 -13244.62,E2 -13244.62} C_VEL
LIN {X 0,Y 361.952,Z 167.398,A -85,B 0,C 180,E1 -13248.1,E2 -13248.1} C_VEL
LIN {X 0,Y 361.888,Z 167.409,A -85,B 0,C 180,E1 -13251.653,E2 -13251.653} C_VEL
LIN {X 0,Y 361.925,Z 167.404,A -85,B 0,C 180,E1 -13255.29,E2 -13255.29} C_VEL
LIN {X 0,Y 361.905,Z 167.405,A -85,B 0,C 180,E1 -13257.779,E2 -13257.779} C_VEL
LIN {X 0,Y 361.834,Z 167.414,A -85,B 0,C 180,E1 -13261.63,E2 -13261.63} C_VEL
LIN {X 0,Y 361.871,Z 167.411,A -85,B 0,C 180,E1 -13265.345,E2 -13265.345} C_VEL
LIN {X 0,Y 361.867,Z 167.41,A -85,B 0,C 180,E1 -13265.48,E2 -13265.48} C_VEL
LIN {X 0,Y 361.187,Z 167.493,A -85,B 0,C 180,E1 -13266.407,E2 -13266.407} C_VEL
LIN {X 0,Y 358.312,Z 167.85,A -85,B 0,C 180,E1 -13267.916,E2 -13267.916} C_VEL
LIN {X 0,Y 355.887,Z 168.157,A -85,B 0,C 180,E1 -13269.136,E2 -13269.136} C_VEL
LIN {X 0,Y 354.854,Z 168.281,A -85,B 0,C 180,E1 -13270.08,E2 -13270.08} C_VEL
LIN {X 0,Y 354.774,Z 168.291,A -85,B 0,C 180,E1 -13270.4,E2 -13270.4} C_VEL
LIN {X 0,Y 354.773,Z 168.29,A -85,B 0,C 180,E1 -13273.895,E2 -13273.895} C_VEL
LIN {X 0,Y 354.786,Z 168.293,A -85,B 0,C 180,E1 -13277.133,E2 -13277.133} C_VEL
LIN {X 0,Y 354.813,Z 168.289,A -85,B 0,C 180,E1 -13280.667,E2 -13280.667} C_VEL
LIN {X 0,Y 354.82,Z 168.286,A -85,B 0,C 180,E1 -13284.301,E2 -13284.301} C_VEL
LIN {X 0,Y 354.785,Z 168.289,A -85,B 0,C 180,E1 -13287.667,E2 -13287.667} C_VEL
LIN {X 0,Y 354.845,Z 168.282,A -85,B 0,C 180,E1 -13291.619,E2 -13291.619} C_VEL
LIN {X 0,Y 354.898,Z 168.277,A -85,B 0,C 180,E1 -13294.173,E2 -13294.173} C_VEL
LIN {X 0,Y 354.835,Z 168.284,A -85,B 0,C 180,E1 -13297.895,E2 -13297.895} C_VEL
LIN {X 0,Y 354.922,Z 168.273,A -85,B 0,C 180,E1 -13301.892,E2 -13301.892} C_VEL
LIN {X 0,Y 354.943,Z 168.272,A -85,B 0,C 180,E1 -13305.982,E2 -13305.982} C_VEL
LIN {X 0,Y 354.978,Z 168.266,A -85,B 0,C 180,E1 -13309.737,E2 -13309.737} C_VEL
LIN {X 0,Y 355.122,Z 168.247,A -85,B 0,C 180,E1 -13313.181,E2 -13313.181} C_VEL
LIN {X 0,Y 355.247,Z 168.234,A -85,B 0,C 180,E1 -13317.733,E2 -13317.733} C_VEL
LIN {X 0,Y 355.397,Z 168.218,A -85,B 0,C 180,E1 -13320.001,E2 -13320.001} C_VEL
LIN {X 0,Y 355.245,Z 168.235,A -85,B 0,C 180,E1 -13322.268,E2 -13322.268} C_VEL
LIN {X 0,Y 355.102,Z 168.25,A -85,B 0,C 180,E1 -13326.82,E2 -13326.82} C_VEL
LIN {X 0,Y 354.958,Z 168.269,A -85,B 0,C 180,E1 -13330.265,E2 -13330.265} C_VEL
LIN {X 0,Y 354.945,Z 168.273,A -85,B 0,C 180,E1 -13334.019,E2 -13334.019} C_VEL
LIN {X 0,Y 354.925,Z 168.274,A -85,B 0,C 180,E1 -13338.109,E2 -13338.109} C_VEL
LIN {X 0,Y 354.837,Z 168.284,A -85,B 0,C 180,E1 -13342.106,E2 -13342.106} C_VEL
LIN {X 0,Y 354.901,Z 168.277,A -85,B 0,C 180,E1 -13345.828,E2 -13345.828} C_VEL
LIN {X 0,Y 354.82,Z 168.288,A -85,B 0,C 180,E1 -13349.682,E2 -13349.682} C_VEL
LIN {X 0,Y 354.808,Z 168.289,A -85,B 0,C 180,E1 -13353.702,E2 -13353.702} C_VEL
LIN {X 0,Y 354.799,Z 168.287,A -85,B 0,C 180,E1 -13356.46,E2 -13356.46} C_VEL
LIN {X 0,Y 354.826,Z 168.288,A -85,B 0,C 180,E1 -13359.424,E2 -13359.424} C_VEL
LIN {X 0,Y 354.819,Z 168.32,A -85,B 0,C 180,E1 -13363.468,E2 -13363.468} C_VEL
LIN {X 0,Y 355.815,Z 173.724,A -85,B 0,C 180,E1 -13366.956,E2 -13366.956} C_VEL
LIN {X 0,Y 356.792,Z 179.036,A -85,B 0,C 180,E1 -13370.194,E2 -13370.194} C_VEL
LIN {X 0,Y 357.387,Z 182.922,A -85,B 0,C 180,E1 -13372.438,E2 -13372.438} C_VEL
LIN {X 0,Y 357.332,Z 186.737,A -85,B 0,C 180,E1 -13374.535,E2 -13374.535} C_VEL
LIN {X 0,Y 356.648,Z 193.257,A -85,B 0,C 180,E1 -13377.925,E2 -13377.925} C_VEL
LIN {X 0,Y 355.817,Z 200.758,A -85,B 0,C 180,E1 -13381.703,E2 -13381.703} C_VEL
LIN {X 0,Y 355.021,Z 208.722,A -85,B 0,C 180,E1 -13385.592,E2 -13385.592} C_VEL
LIN {X 0,Y 354.426,Z 216.688,A -85,B 0,C 180,E1 -13389.392,E2 -13389.392} C_VEL
LIN {X 0,Y 354.398,Z 217.286,A -85,B 0,C 180,E1 -13389.675,E2 -13389.675} C_VEL
LIN {X 0,Y 356.769,Z 231.399,A -85,B 0,C 180,E1 -13390.322,E2 -13390.322} C_VEL
LIN {X 0,Y 358.46,Z 244.315,A -85,B 0,C 180,E1 -13391.134,E2 -13391.134} C_VEL
LIN {X 0,Y 359.543,Z 256.113,A -85,B 0,C 180,E1 -13392.069,E2 -13392.069} C_VEL
LIN {X 0,Y 358.403,Z 266.781,A -85,B 0,C 180,E1 -13393.041,E2 -13393.041} C_VEL
LIN {X 0,Y 357.342,Z 277.327,A -85,B 0,C 180,E1 -13394.252,E2 -13394.252} C_VEL
LIN {X 0,Y 356.349,Z 287.606,A -85,B 0,C 180,E1 -13395.728,E2 -13395.728} C_VEL
LIN {X 0,Y 355.449,Z 295.689,A -85,B 0,C 180,E1 -13397.148,E2 -13397.148} C_VEL
LIN {X 0,Y 354.557,Z 303.627,A -85,B 0,C 180,E1 -13398.857,E2 -13398.857} C_VEL
LIN {X 0,Y 354.088,Z 309.011,A -85,B 0,C 180,E1 -13400.287,E2 -13400.287} C_VEL
LIN {X 0,Y 353.654,Z 314.275,A -85,B 0,C 180,E1 -13402.004,E2 -13402.004} C_VEL
LIN {X 0,Y 353.436,Z 318.628,A -85,B 0,C 180,E1 -13403.851,E2 -13403.851} C_VEL
LIN {X 0,Y 353.358,Z 321.377,A -85,B 0,C 180,E1 -13405.437,E2 -13405.437} C_VEL
LIN {X 0,Y 353.275,Z 322.84,A -85,B 0,C 180,E1 -13406.579,E2 -13406.579} C_VEL
LIN {X 0,Y 353.316,Z 323.866,A -85,B 0,C 180,E1 -13407.72,E2 -13407.72} C_VEL
LIN {X 0,Y 353.395,Z 324.497,A -85,B 0,C 180,E1 -13408.861,E2 -13408.861} C_VEL
LIN {X 0,Y 353.404,Z 324.73,A -85,B 0,C 180,E1 -13410,E2 -13410} C_VEL
LIN {X 0,Y 353.393,Z 324.54,A -85,B 0,C 180,E1 -13411.14,E2 -13411.14} C_VEL
LIN {X 0,Y 353.281,Z 322.902,A -85,B 0,C 180,E1 -13413.422,E2 -13413.422} C_VEL
LIN {X 0,Y 353.338,Z 321.491,A -85,B 0,C 180,E1 -13414.564,E2 -13414.564} C_VEL
LIN {X 0,Y 353.437,Z 318.775,A -85,B 0,C 180,E1 -13416.149,E2 -13416.149} C_VEL
LIN {X 0,Y 353.655,Z 314.522,A -85,B 0,C 180,E1 -13417.996,E2 -13417.996} C_VEL
LIN {X 0,Y 354.201,Z 308.411,A -85,B 0,C 180,E1 -13419.998,E2 -13419.998} C_VEL
LIN {X 0,Y 354.857,Z 301.727,A -85,B 0,C 180,E1 -13421.713,E2 -13421.713} C_VEL
LIN {X 0,Y 355.835,Z 293.472,A -85,B 0,C 180,E1 -13423.419,E2 -13423.419} C_VEL
